   1:  PR[GP1:91,1] = PR[GP1:90,1] + -74.339;
   1:  PR[GP1:91,2] = PR[GP1:90,2] + 0.256;
   1:L PR[91] 10mm/sec CNT100;
   1:  PR[GP1:91,1] = PR[GP1:90,1] + -74.139;
   1:  PR[GP1:91,2] = PR[GP1:90,2] + -1.545;
   1:L PR[91] 10mm/sec CNT100;
   1:  PR[GP1:91,1] = PR[GP1:90,1] + -72.276;
   1:  PR[GP1:91,2] = PR[GP1:90,2] + -11.283;
   1:L PR[91] 10mm/sec CNT100;
   1:  PR[GP1:91,1] = PR[GP1:90,1] + -71.760;
   1:  PR[GP1:91,2] = PR[GP1:90,2] + -12.778;
   1:L PR[91] 10mm/sec CNT100;
   1:  PR[GP1:91,1] = PR[GP1:90,1] + -70.908;
   1:  PR[GP1:91,2] = PR[GP1:90,2] + -14.156;
   1:L PR[91] 10mm/sec CNT100;
   1:  PR[GP1:91,1] = PR[GP1:90,1] + -65.415;
   1:  PR[GP1:91,2] = PR[GP1:90,2] + -22.829;
   1:L PR[91] 10mm/sec CNT100;
   1:  PR[GP1:91,1] = PR[GP1:90,1] + -64.501;
   1:  PR[GP1:91,2] = PR[GP1:90,2] + -23.762;
   1:L PR[91] 10mm/sec CNT100;
   1:  PR[GP1:91,1] = PR[GP1:90,1] + -63.337;
   1:  PR[GP1:91,2] = PR[GP1:90,2] + -24.515;
   1:L PR[91] 10mm/sec CNT100;
   1:  PR[GP1:91,1] = PR[GP1:90,1] + -54.747;
   1:  PR[GP1:91,2] = PR[GP1:90,2] + -30.797;
   1:L PR[91] 10mm/sec CNT100;
   1:  PR[GP1:91,1] = PR[GP1:90,1] + -53.911;
   1:  PR[GP1:91,2] = PR[GP1:90,2] + -31.105;
   1:L PR[91] 10mm/sec CNT100;
   1:  PR[GP1:91,1] = PR[GP1:90,1] + -42.471;
   1:  PR[GP1:91,2] = PR[GP1:90,2] + -34.073;
   1:L PR[91] 10mm/sec CNT100;
   1:  PR[GP1:91,1] = PR[GP1:90,1] + -42.174;
   1:  PR[GP1:91,2] = PR[GP1:90,2] + -34.112;
   1:L PR[91] 10mm/sec CNT100;
   1:  PR[GP1:91,1] = PR[GP1:90,1] + -41.849;
   1:  PR[GP1:91,2] = PR[GP1:90,2] + -34.082;
   1:L PR[91] 10mm/sec CNT100;
   1:  PR[GP1:91,1] = PR[GP1:90,1] + -34.975;
   1:  PR[GP1:91,2] = PR[GP1:90,2] + -33.253;
   1:L PR[91] 10mm/sec CNT100;
   1:  PR[GP1:91,1] = PR[GP1:90,1] + -29.454;
   1:  PR[GP1:91,2] = PR[GP1:90,2] + -32.634;
   1:L PR[91] 10mm/sec CNT100;
   1:  PR[GP1:91,1] = PR[GP1:90,1] + -28.961;
   1:  PR[GP1:91,2] = PR[GP1:90,2] + -32.418;
   1:L PR[91] 10mm/sec CNT100;
   1:  PR[GP1:91,1] = PR[GP1:90,1] + -18.207;
   1:  PR[GP1:91,2] = PR[GP1:90,2] + -26.771;
   1:L PR[91] 10mm/sec CNT100;
   1:  PR[GP1:91,1] = PR[GP1:90,1] + -16.790;
   1:  PR[GP1:91,2] = PR[GP1:90,2] + -25.386;
   1:L PR[91] 10mm/sec CNT100;
   1:  PR[GP1:91,1] = PR[GP1:90,1] + -9.851;
   1:  PR[GP1:91,2] = PR[GP1:90,2] + -17.341;
   1:L PR[91] 10mm/sec CNT100;
   1:  PR[GP1:91,1] = PR[GP1:90,1] + -8.556;
   1:  PR[GP1:91,2] = PR[GP1:90,2] + -14.548;
   1:L PR[91] 10mm/sec CNT100;
   1:  PR[GP1:91,1] = PR[GP1:90,1] + -5.279;
   1:  PR[GP1:91,2] = PR[GP1:90,2] + -5.083;
   1:L PR[91] 10mm/sec CNT100;
   1:  PR[GP1:91,1] = PR[GP1:90,1] + 4.751;
   1:L PR[91] 10mm/sec CNT100;
   1:  PR[GP1:91,1] = PR[GP1:90,1] + 7.580;
   1:  PR[GP1:91,2] = PR[GP1:90,2] + -13.769;
   1:  PR[GP1:91,3] = PR[GP1:90,3] + 17.995;
   1:L PR[91] 10mm/sec CNT100;
   1:  PR[GP1:91,1] = PR[GP1:90,1] + 9.344;
   1:  PR[GP1:91,2] = PR[GP1:90,2] + -17.567;
   1:L PR[91] 10mm/sec CNT100;
   1:  PR[GP1:91,1] = PR[GP1:90,1] + 15.538;
   1:  PR[GP1:91,2] = PR[GP1:90,2] + -24.755;
   1:L PR[91] 10mm/sec CNT100;
   1:  PR[GP1:91,1] = PR[GP1:90,1] + 17.739;
   1:  PR[GP1:91,2] = PR[GP1:90,2] + -26.911;
   1:L PR[91] 10mm/sec CNT100;
   1:  PR[GP1:91,1] = PR[GP1:90,1] + 27.542;
   1:  PR[GP1:91,2] = PR[GP1:90,2] + -32.059;
   1:L PR[91] 10mm/sec CNT100;
   1:  PR[GP1:91,1] = PR[GP1:90,1] + 28.984;
   1:  PR[GP1:91,2] = PR[GP1:90,2] + -32.692;
   1:L PR[91] 10mm/sec CNT100;
   1:  PR[GP1:91,1] = PR[GP1:90,1] + 41.685;
   1:  PR[GP1:91,2] = PR[GP1:90,2] + -34.108;
   1:L PR[91] 10mm/sec CNT100;
   1:  PR[GP1:91,1] = PR[GP1:90,1] + 53.747;
   1:  PR[GP1:91,2] = PR[GP1:90,2] + -30.970;
   1:L PR[91] 10mm/sec CNT100;
   1:  PR[GP1:91,1] = PR[GP1:90,1] + 54.176;
   1:  PR[GP1:91,2] = PR[GP1:90,2] + -30.813;
   1:L PR[91] 10mm/sec CNT100;
   1:  PR[GP1:91,1] = PR[GP1:90,1] + 54.570;
   1:  PR[GP1:91,2] = PR[GP1:90,2] + -30.558;
   1:L PR[91] 10mm/sec CNT100;
   1:  PR[GP1:91,1] = PR[GP1:90,1] + 64.128;
   1:  PR[GP1:91,2] = PR[GP1:90,2] + -23.600;
   1:L PR[91] 10mm/sec CNT100;
   1:  PR[GP1:91,1] = PR[GP1:90,1] + 64.755;
   1:  PR[GP1:91,2] = PR[GP1:90,2] + -22.960;
   1:L PR[91] 10mm/sec CNT100;
   1:  PR[GP1:91,1] = PR[GP1:90,1] + 65.254;
   1:  PR[GP1:91,2] = PR[GP1:90,2] + -22.153;
   1:L PR[91] 10mm/sec CNT100;
   1:  PR[GP1:91,1] = PR[GP1:90,1] + 71.263;
   1:  PR[GP1:91,2] = PR[GP1:90,2] + -12.665;
   1:L PR[91] 10mm/sec CNT100;
   1:  PR[GP1:91,1] = PR[GP1:90,1] + 71.637;
   1:  PR[GP1:91,2] = PR[GP1:90,2] + -11.579;
   1:L PR[91] 10mm/sec CNT100;
   1:  PR[GP1:91,1] = PR[GP1:90,1] + 71.774;
   1:  PR[GP1:91,2] = PR[GP1:90,2] + -10.346;
   1:L PR[91] 10mm/sec CNT100;
   1:  PR[GP1:91,1] = PR[GP1:90,1] + 73.791;
   1:  PR[GP1:91,2] = PR[GP1:90,2] + 0.302;
   1:L PR[91] 10mm/sec CNT100;
   1:  PR[GP1:91,1] = PR[GP1:90,1] + 73.634;
   1:  PR[GP1:91,2] = PR[GP1:90,2] + 1.715;
   1:L PR[91] 10mm/sec CNT100;
   1:  PR[GP1:91,1] = PR[GP1:90,1] + 71.645;
   1:  PR[GP1:91,2] = PR[GP1:90,2] + 12.115;
   1:L PR[91] 10mm/sec CNT100;
   1:  PR[GP1:91,1] = PR[GP1:90,1] + 71.262;
   1:  PR[GP1:91,2] = PR[GP1:90,2] + 13.226;
   1:L PR[91] 10mm/sec CNT100;
   1:  PR[GP1:91,1] = PR[GP1:90,1] + 70.623;
   1:  PR[GP1:91,2] = PR[GP1:90,2] + 14.259;
   1:L PR[91] 10mm/sec CNT100;
   1:  PR[GP1:91,1] = PR[GP1:90,1] + 64.757;
   1:  PR[GP1:91,2] = PR[GP1:90,2] + 23.516;
   1:L PR[91] 10mm/sec CNT100;
   1:  PR[GP1:91,1] = PR[GP1:90,1] + 64.140;
   1:  PR[GP1:91,2] = PR[GP1:90,2] + 24.146;
   1:L PR[91] 10mm/sec CNT100;
   1:  PR[GP1:91,1] = PR[GP1:90,1] + 63.331;
   1:  PR[GP1:91,2] = PR[GP1:90,2] + 24.669;
   1:L PR[91] 10mm/sec CNT100;
   1:  PR[GP1:91,1] = PR[GP1:90,1] + 54.159;
   1:  PR[GP1:91,2] = PR[GP1:90,2] + 31.377;
   1:L PR[91] 10mm/sec CNT100;
   1:  PR[GP1:91,1] = PR[GP1:90,1] + 53.747;
   1:  PR[GP1:91,2] = PR[GP1:90,2] + 31.529;
   1:L PR[91] 10mm/sec CNT100;
   1:  PR[GP1:91,1] = PR[GP1:90,1] + 41.668;
   1:  PR[GP1:91,2] = PR[GP1:90,2] + 34.670;
   1:L PR[91] 10mm/sec CNT100;
   1:  PR[GP1:91,1] = PR[GP1:90,1] + 41.604;
   1:  PR[GP1:91,2] = PR[GP1:90,2] + 34.667;
   1:L PR[91] 10mm/sec CNT100;
   1:  PR[GP1:91,1] = PR[GP1:90,1] + 28.984;
   1:  PR[GP1:91,2] = PR[GP1:90,2] + 33.250;
   1:L PR[91] 10mm/sec CNT100;
   1:  PR[GP1:91,1] = PR[GP1:90,1] + 27.542;
   1:  PR[GP1:91,2] = PR[GP1:90,2] + 32.617;
   1:L PR[91] 10mm/sec CNT100;
   1:  PR[GP1:91,1] = PR[GP1:90,1] + 17.739;
   1:  PR[GP1:91,2] = PR[GP1:90,2] + 27.469;
   1:L PR[91] 10mm/sec CNT100;
   1:  PR[GP1:91,1] = PR[GP1:90,1] + 15.538;
   1:  PR[GP1:91,2] = PR[GP1:90,2] + 25.313;
   1:L PR[91] 10mm/sec CNT100;
   1:  PR[GP1:91,1] = PR[GP1:90,1] + 9.344;
   1:  PR[GP1:91,2] = PR[GP1:90,2] + 18.125;
   1:L PR[91] 10mm/sec CNT100;
   1:  PR[GP1:91,1] = PR[GP1:90,1] + 7.579;
   1:  PR[GP1:91,2] = PR[GP1:90,2] + 14.325;
   1:L PR[91] 10mm/sec CNT100;
   1:  PR[GP1:91,1] = PR[GP1:90,1] + 4.686;
   1:  PR[GP1:91,2] = PR[GP1:90,2] + 5.966;
   1:L PR[91] 10mm/sec CNT100;
   1:  PR[GP1:91,1] = PR[GP1:90,1] + -5.214;
   1:L PR[91] 10mm/sec CNT100;
   1:  PR[GP1:91,1] = PR[GP1:90,1] + -8.111;
   1:  PR[GP1:91,2] = PR[GP1:90,2] + 14.333;
   1:L PR[91] 10mm/sec CNT100;
   1:  PR[GP1:91,1] = PR[GP1:90,1] + -9.876;
   1:  PR[GP1:91,2] = PR[GP1:90,2] + 18.139;
   1:L PR[91] 10mm/sec CNT100;
   1:  PR[GP1:91,1] = PR[GP1:90,1] + -16.071;
   1:  PR[GP1:91,2] = PR[GP1:90,2] + 25.322;
   1:L PR[91] 10mm/sec CNT100;
   1:  PR[GP1:91,1] = PR[GP1:90,1] + -18.271;
   1:  PR[GP1:91,2] = PR[GP1:90,2] + 27.472;
   1:L PR[91] 10mm/sec CNT100;
   1:  PR[GP1:91,1] = PR[GP1:90,1] + -28.075;
   1:  PR[GP1:91,2] = PR[GP1:90,2] + 32.620;
   1:L PR[91] 10mm/sec CNT100;
   1:  PR[GP1:91,1] = PR[GP1:90,1] + -29.516;
   1:  PR[GP1:91,2] = PR[GP1:90,2] + 33.252;
   1:L PR[91] 10mm/sec CNT100;
   1:  PR[GP1:91,1] = PR[GP1:90,1] + -42.215;
   1:  PR[GP1:91,2] = PR[GP1:90,2] + 34.666;
   1:L PR[91] 10mm/sec CNT100;
   1:  PR[GP1:91,1] = PR[GP1:90,1] + -54.276;
   1:  PR[GP1:91,2] = PR[GP1:90,2] + 31.527;
   1:L PR[91] 10mm/sec CNT100;
   1:  PR[GP1:91,1] = PR[GP1:90,1] + -54.705;
   1:  PR[GP1:91,2] = PR[GP1:90,2] + 31.369;
   1:L PR[91] 10mm/sec CNT100;
   1:  PR[GP1:91,1] = PR[GP1:90,1] + -55.099;
   1:  PR[GP1:91,2] = PR[GP1:90,2] + 31.114;
   1:L PR[91] 10mm/sec CNT100;
   1:  PR[GP1:91,1] = PR[GP1:90,1] + -64.656;
   1:  PR[GP1:91,2] = PR[GP1:90,2] + 24.157;
   1:L PR[91] 10mm/sec CNT100;
   1:  PR[GP1:91,1] = PR[GP1:90,1] + -65.285;
   1:  PR[GP1:91,2] = PR[GP1:90,2] + 23.515;
   1:L PR[91] 10mm/sec CNT100;
   1:  PR[GP1:91,1] = PR[GP1:90,1] + -71.790;
   1:  PR[GP1:91,2] = PR[GP1:90,2] + 13.220;
   1:L PR[91] 10mm/sec CNT100;
   1:  PR[GP1:91,1] = PR[GP1:90,1] + -72.164;
   1:  PR[GP1:91,2] = PR[GP1:90,2] + 12.134;
   1:L PR[91] 10mm/sec CNT100;
   1:  PR[GP1:91,1] = PR[GP1:90,1] + -72.301;
   1:  PR[GP1:91,2] = PR[GP1:90,2] + 10.901;
   1:L PR[91] 10mm/sec CNT100;
   1:  PR[GP1:91,1] = PR[GP1:90,1] + -74.318;
   1:  PR[GP1:91,2] = PR[GP1:90,2] + 0.256;
   1:L PR[91] 10mm/sec CNT100;
   1:  PR[GP1:91,1] = PR[GP1:90,1] + -74.160;
   1:  PR[GP1:91,2] = PR[GP1:90,2] + -1.157;
   1:L PR[91] 10mm/sec CNT100;
   1:  PR[GP1:91,1] = PR[GP1:90,1] + -72.172;
   1:  PR[GP1:91,2] = PR[GP1:90,2] + -11.554;
   1:L PR[91] 10mm/sec CNT100;
   1:  PR[GP1:91,1] = PR[GP1:90,1] + -71.789;
   1:  PR[GP1:91,2] = PR[GP1:90,2] + -12.665;
   1:L PR[91] 10mm/sec CNT100;
   1:  PR[GP1:91,1] = PR[GP1:90,1] + -71.150;
   1:  PR[GP1:91,2] = PR[GP1:90,2] + -13.698;
   1:L PR[91] 10mm/sec CNT100;
   1:  PR[GP1:91,1] = PR[GP1:90,1] + -65.285;
   1:  PR[GP1:91,2] = PR[GP1:90,2] + -22.957;
   1:L PR[91] 10mm/sec CNT100;
   1:  PR[GP1:91,1] = PR[GP1:90,1] + -64.667;
   1:  PR[GP1:91,2] = PR[GP1:90,2] + -23.587;
   1:L PR[91] 10mm/sec CNT100;
   1:  PR[GP1:91,1] = PR[GP1:90,1] + -63.859;
   1:  PR[GP1:91,2] = PR[GP1:90,2] + -24.110;
   1:L PR[91] 10mm/sec CNT100;
   1:  PR[GP1:91,1] = PR[GP1:90,1] + -54.688;
   1:  PR[GP1:91,2] = PR[GP1:90,2] + -30.818;
   1:L PR[91] 10mm/sec CNT100;
   1:  PR[GP1:91,1] = PR[GP1:90,1] + -54.276;
   1:  PR[GP1:91,2] = PR[GP1:90,2] + -30.969;
   1:L PR[91] 10mm/sec CNT100;
   1:  PR[GP1:91,1] = PR[GP1:90,1] + -42.215;
   1:  PR[GP1:91,2] = PR[GP1:90,2] + -34.107;
   1:L PR[91] 10mm/sec CNT100;
   1:  PR[GP1:91,1] = PR[GP1:90,1] + -29.516;
   1:  PR[GP1:91,2] = PR[GP1:90,2] + -32.694;
   1:L PR[91] 10mm/sec CNT100;
   1:  PR[GP1:91,1] = PR[GP1:90,1] + -28.075;
   1:  PR[GP1:91,2] = PR[GP1:90,2] + -32.062;
   1:L PR[91] 10mm/sec CNT100;
   1:  PR[GP1:91,1] = PR[GP1:90,1] + -18.271;
   1:  PR[GP1:91,2] = PR[GP1:90,2] + -26.914;
   1:L PR[91] 10mm/sec CNT100;
   1:  PR[GP1:91,1] = PR[GP1:90,1] + -16.071;
   1:  PR[GP1:91,2] = PR[GP1:90,2] + -24.763;
   1:L PR[91] 10mm/sec CNT100;
   1:  PR[GP1:91,1] = PR[GP1:90,1] + -9.876;
   1:  PR[GP1:91,2] = PR[GP1:90,2] + -17.581;
   1:L PR[91] 10mm/sec CNT100;
   1:  PR[GP1:91,1] = PR[GP1:90,1] + -8.110;
   1:  PR[GP1:91,2] = PR[GP1:90,2] + -13.773;
   1:L PR[91] 10mm/sec CNT100;
   1:  PR[GP1:91,1] = PR[GP1:90,1] + -5.214;
   1:  PR[GP1:91,2] = PR[GP1:90,2] + -5.408;
   1:L PR[91] 10mm/sec CNT100;
   1:  PR[GP1:91,1] = PR[GP1:90,1] + 4.686;
   1:L PR[91] 10mm/sec CNT100;
   1:  PR[GP1:91,1] = PR[GP1:90,1] + 7.134;
   1:  PR[GP1:91,2] = PR[GP1:90,2] + -12.995;
   1:  PR[GP1:91,3] = PR[GP1:90,3] + 18.605;
   1:L PR[91] 10mm/sec CNT100;
   1:  PR[GP1:91,1] = PR[GP1:90,1] + 9.368;
   1:  PR[GP1:91,2] = PR[GP1:90,2] + -17.806;
   1:L PR[91] 10mm/sec CNT100;
   1:  PR[GP1:91,1] = PR[GP1:90,1] + 14.818;
   1:  PR[GP1:91,2] = PR[GP1:90,2] + -24.130;
   1:L PR[91] 10mm/sec CNT100;
   1:  PR[GP1:91,1] = PR[GP1:90,1] + 17.802;
   1:  PR[GP1:91,2] = PR[GP1:90,2] + -27.054;
   1:L PR[91] 10mm/sec CNT100;
   1:  PR[GP1:91,1] = PR[GP1:90,1] + 26.655;
   1:  PR[GP1:91,2] = PR[GP1:90,2] + -31.703;
   1:L PR[91] 10mm/sec CNT100;
   1:  PR[GP1:91,1] = PR[GP1:90,1] + 29.045;
   1:  PR[GP1:91,2] = PR[GP1:90,2] + -32.752;
   1:L PR[91] 10mm/sec CNT100;
   1:  PR[GP1:91,1] = PR[GP1:90,1] + 40.686;
   1:  PR[GP1:91,2] = PR[GP1:90,2] + -34.059;
   1:L PR[91] 10mm/sec CNT100;
   1:  PR[GP1:91,1] = PR[GP1:90,1] + 41.701;
   1:  PR[GP1:91,2] = PR[GP1:90,2] + -34.116;
   1:L PR[91] 10mm/sec CNT100;
   1:  PR[GP1:91,1] = PR[GP1:90,1] + 54.124;
   1:  PR[GP1:91,2] = PR[GP1:90,2] + -30.822;
   1:L PR[91] 10mm/sec CNT100;
   1:  PR[GP1:91,1] = PR[GP1:90,1] + 64.295;
   1:  PR[GP1:91,2] = PR[GP1:90,2] + -23.426;
   1:L PR[91] 10mm/sec CNT100;
   1:  PR[GP1:91,1] = PR[GP1:90,1] + 64.627;
   1:  PR[GP1:91,2] = PR[GP1:90,2] + -23.086;
   1:L PR[91] 10mm/sec CNT100;
   1:  PR[GP1:91,1] = PR[GP1:90,1] + 71.291;
   1:  PR[GP1:91,2] = PR[GP1:90,2] + -12.552;
   1:L PR[91] 10mm/sec CNT100;
   1:  PR[GP1:91,1] = PR[GP1:90,1] + 71.533;
   1:  PR[GP1:91,2] = PR[GP1:90,2] + -11.850;
   1:L PR[91] 10mm/sec CNT100;
   1:  PR[GP1:91,1] = PR[GP1:90,1] + 71.625;
   1:  PR[GP1:91,2] = PR[GP1:90,2] + -11.021;
   1:L PR[91] 10mm/sec CNT100;
   1:  PR[GP1:91,1] = PR[GP1:90,1] + 73.770;
   1:  PR[GP1:91,2] = PR[GP1:90,2] + 0.302;
   1:L PR[91] 10mm/sec CNT100;
   1:  PR[GP1:91,1] = PR[GP1:90,1] + 73.656;
   1:  PR[GP1:91,2] = PR[GP1:90,2] + 1.327;
   1:L PR[91] 10mm/sec CNT100;
   1:  PR[GP1:91,1] = PR[GP1:90,1] + 71.541;
   1:  PR[GP1:91,2] = PR[GP1:90,2] + 12.386;
   1:L PR[91] 10mm/sec CNT100;
   1:  PR[GP1:91,1] = PR[GP1:90,1] + 71.291;
   1:  PR[GP1:91,2] = PR[GP1:90,2] + 13.110;
   1:L PR[91] 10mm/sec CNT100;
   1:  PR[GP1:91,1] = PR[GP1:90,1] + 64.627;
   1:  PR[GP1:91,2] = PR[GP1:90,2] + 23.644;
   1:L PR[91] 10mm/sec CNT100;
   1:  PR[GP1:91,1] = PR[GP1:90,1] + 64.306;
   1:  PR[GP1:91,2] = PR[GP1:90,2] + 23.972;
   1:L PR[91] 10mm/sec CNT100;
   1:  PR[GP1:91,1] = PR[GP1:90,1] + 63.853;
   1:  PR[GP1:91,2] = PR[GP1:90,2] + 24.265;
   1:L PR[91] 10mm/sec CNT100;
   1:  PR[GP1:91,1] = PR[GP1:90,1] + 54.123;
   1:  PR[GP1:91,2] = PR[GP1:90,2] + 31.380;
   1:L PR[91] 10mm/sec CNT100;
   1:  PR[GP1:91,1] = PR[GP1:90,1] + 41.701;
   1:  PR[GP1:91,2] = PR[GP1:90,2] + 34.674;
   1:L PR[91] 10mm/sec CNT100;
   1:  PR[GP1:91,1] = PR[GP1:90,1] + 40.686;
   1:  PR[GP1:91,2] = PR[GP1:90,2] + 34.617;
   1:L PR[91] 10mm/sec CNT100;
   1:  PR[GP1:91,1] = PR[GP1:90,1] + 29.045;
   1:  PR[GP1:91,2] = PR[GP1:90,2] + 33.310;
   1:L PR[91] 10mm/sec CNT100;
   1:  PR[GP1:91,1] = PR[GP1:90,1] + 26.655;
   1:  PR[GP1:91,2] = PR[GP1:90,2] + 32.261;
   1:L PR[91] 10mm/sec CNT100;
   1:  PR[GP1:91,1] = PR[GP1:90,1] + 17.802;
   1:  PR[GP1:91,2] = PR[GP1:90,2] + 27.612;
   1:L PR[91] 10mm/sec CNT100;
   1:  PR[GP1:91,1] = PR[GP1:90,1] + 14.818;
   1:  PR[GP1:91,2] = PR[GP1:90,2] + 24.688;
   1:L PR[91] 10mm/sec CNT100;
   1:  PR[GP1:91,1] = PR[GP1:90,1] + 9.368;
   1:  PR[GP1:91,2] = PR[GP1:90,2] + 18.364;
   1:L PR[91] 10mm/sec CNT100;
   1:  PR[GP1:91,1] = PR[GP1:90,1] + 7.133;
   1:  PR[GP1:91,2] = PR[GP1:90,2] + 13.550;
   1:L PR[91] 10mm/sec CNT100;
   1:  PR[GP1:91,1] = PR[GP1:90,1] + 4.620;
   1:  PR[GP1:91,2] = PR[GP1:90,2] + 6.291;
   1:L PR[91] 10mm/sec CNT100;
   1:  PR[GP1:91,1] = PR[GP1:90,1] + -5.149;
   1:L PR[91] 10mm/sec CNT100;
   1:  PR[GP1:91,1] = PR[GP1:90,1] + -7.665;
   1:  PR[GP1:91,2] = PR[GP1:90,2] + 13.559;
   1:L PR[91] 10mm/sec CNT100;
   1:  PR[GP1:91,1] = PR[GP1:90,1] + -9.901;
   1:  PR[GP1:91,2] = PR[GP1:90,2] + 18.379;
   1:L PR[91] 10mm/sec CNT100;
   1:  PR[GP1:91,1] = PR[GP1:90,1] + -15.352;
   1:  PR[GP1:91,2] = PR[GP1:90,2] + 24.699;
   1:L PR[91] 10mm/sec CNT100;
   1:  PR[GP1:91,1] = PR[GP1:90,1] + -18.335;
   1:  PR[GP1:91,2] = PR[GP1:90,2] + 27.615;
   1:L PR[91] 10mm/sec CNT100;
   1:  PR[GP1:91,1] = PR[GP1:90,1] + -27.189;
   1:  PR[GP1:91,2] = PR[GP1:90,2] + 32.264;
   1:L PR[91] 10mm/sec CNT100;
   1:  PR[GP1:91,1] = PR[GP1:90,1] + -29.577;
   1:  PR[GP1:91,2] = PR[GP1:90,2] + 33.313;
   1:L PR[91] 10mm/sec CNT100;
   1:  PR[GP1:91,1] = PR[GP1:90,1] + -41.217;
   1:  PR[GP1:91,2] = PR[GP1:90,2] + 34.617;
   1:L PR[91] 10mm/sec CNT100;
   1:  PR[GP1:91,1] = PR[GP1:90,1] + -42.231;
   1:  PR[GP1:91,2] = PR[GP1:90,2] + 34.673;
   1:L PR[91] 10mm/sec CNT100;
   1:  PR[GP1:91,1] = PR[GP1:90,1] + -54.653;
   1:  PR[GP1:91,2] = PR[GP1:90,2] + 31.379;
   1:L PR[91] 10mm/sec CNT100;
   1:  PR[GP1:91,1] = PR[GP1:90,1] + -64.822;
   1:  PR[GP1:91,2] = PR[GP1:90,2] + 23.983;
   1:L PR[91] 10mm/sec CNT100;
   1:  PR[GP1:91,1] = PR[GP1:90,1] + -65.155;
   1:  PR[GP1:91,2] = PR[GP1:90,2] + 23.643;
   1:L PR[91] 10mm/sec CNT100;
   1:  PR[GP1:91,1] = PR[GP1:90,1] + -71.818;
   1:  PR[GP1:91,2] = PR[GP1:90,2] + 13.107;
   1:L PR[91] 10mm/sec CNT100;
   1:  PR[GP1:91,1] = PR[GP1:90,1] + -72.060;
   1:  PR[GP1:91,2] = PR[GP1:90,2] + 12.405;
   1:L PR[91] 10mm/sec CNT100;
   1:  PR[GP1:91,1] = PR[GP1:90,1] + -72.152;
   1:  PR[GP1:91,2] = PR[GP1:90,2] + 11.575;
   1:L PR[91] 10mm/sec CNT100;
   1:  PR[GP1:91,1] = PR[GP1:90,1] + -74.296;
   1:  PR[GP1:91,2] = PR[GP1:90,2] + 0.256;
   1:L PR[91] 10mm/sec CNT100;
   1:  PR[GP1:91,1] = PR[GP1:90,1] + -74.182;
   1:  PR[GP1:91,2] = PR[GP1:90,2] + -0.769;
   1:L PR[91] 10mm/sec CNT100;
   1:  PR[GP1:91,1] = PR[GP1:90,1] + -72.067;
   1:  PR[GP1:91,2] = PR[GP1:90,2] + -11.825;
   1:L PR[91] 10mm/sec CNT100;
   1:  PR[GP1:91,1] = PR[GP1:90,1] + -71.817;
   1:  PR[GP1:91,2] = PR[GP1:90,2] + -12.551;
   1:L PR[91] 10mm/sec CNT100;
   1:  PR[GP1:91,1] = PR[GP1:90,1] + -71.392;
   1:  PR[GP1:91,2] = PR[GP1:90,2] + -13.239;
   1:L PR[91] 10mm/sec CNT100;
   1:  PR[GP1:91,1] = PR[GP1:90,1] + -65.155;
   1:  PR[GP1:91,2] = PR[GP1:90,2] + -23.085;
   1:L PR[91] 10mm/sec CNT100;
   1:  PR[GP1:91,1] = PR[GP1:90,1] + -64.834;
   1:  PR[GP1:91,2] = PR[GP1:90,2] + -23.413;
   1:L PR[91] 10mm/sec CNT100;
   1:  PR[GP1:91,1] = PR[GP1:90,1] + -64.381;
   1:  PR[GP1:91,2] = PR[GP1:90,2] + -23.706;
   1:L PR[91] 10mm/sec CNT100;
   1:  PR[GP1:91,1] = PR[GP1:90,1] + -54.632;
   1:  PR[GP1:91,2] = PR[GP1:90,2] + -30.836;
   1:L PR[91] 10mm/sec CNT100;
   1:  PR[GP1:91,1] = PR[GP1:90,1] + -42.232;
   1:  PR[GP1:91,2] = PR[GP1:90,2] + -34.115;
   1:L PR[91] 10mm/sec CNT100;
   1:  PR[GP1:91,1] = PR[GP1:90,1] + -41.217;
   1:  PR[GP1:91,2] = PR[GP1:90,2] + -34.059;
   1:L PR[91] 10mm/sec CNT100;
   1:  PR[GP1:91,1] = PR[GP1:90,1] + -29.577;
   1:  PR[GP1:91,2] = PR[GP1:90,2] + -32.755;
   1:L PR[91] 10mm/sec CNT100;
   1:  PR[GP1:91,1] = PR[GP1:90,1] + -27.189;
   1:  PR[GP1:91,2] = PR[GP1:90,2] + -31.706;
   1:L PR[91] 10mm/sec CNT100;
   1:  PR[GP1:91,1] = PR[GP1:90,1] + -18.335;
   1:  PR[GP1:91,2] = PR[GP1:90,2] + -27.057;
   1:L PR[91] 10mm/sec CNT100;
   1:  PR[GP1:91,1] = PR[GP1:90,1] + -15.351;
   1:  PR[GP1:91,2] = PR[GP1:90,2] + -24.141;
   1:L PR[91] 10mm/sec CNT100;
   1:  PR[GP1:91,1] = PR[GP1:90,1] + -9.901;
   1:  PR[GP1:91,2] = PR[GP1:90,2] + -17.821;
   1:L PR[91] 10mm/sec CNT100;
   1:  PR[GP1:91,1] = PR[GP1:90,1] + -7.664;
   1:  PR[GP1:91,2] = PR[GP1:90,2] + -12.997;
   1:L PR[91] 10mm/sec CNT100;
   1:  PR[GP1:91,1] = PR[GP1:90,1] + -5.149;
   1:  PR[GP1:91,2] = PR[GP1:90,2] + -5.733;
   1:L PR[91] 10mm/sec CNT100;
   1:  PR[GP1:91,1] = PR[GP1:90,1] + 4.620;
   1:L PR[91] 10mm/sec CNT100;
   1:  PR[GP1:91,1] = PR[GP1:90,1] + 6.689;
   1:  PR[GP1:91,2] = PR[GP1:90,2] + -12.221;
   1:  PR[GP1:91,3] = PR[GP1:90,3] + 19.215;
   1:L PR[91] 10mm/sec CNT100;
   1:  PR[GP1:91,1] = PR[GP1:90,1] + 9.392;
   1:  PR[GP1:91,2] = PR[GP1:90,2] + -18.045;
   1:L PR[91] 10mm/sec CNT100;
   1:  PR[GP1:91,1] = PR[GP1:90,1] + 14.098;
   1:  PR[GP1:91,2] = PR[GP1:90,2] + -23.505;
   1:L PR[91] 10mm/sec CNT100;
   1:  PR[GP1:91,1] = PR[GP1:90,1] + 17.865;
   1:  PR[GP1:91,2] = PR[GP1:90,2] + -27.197;
   1:L PR[91] 10mm/sec CNT100;
   1:  PR[GP1:91,1] = PR[GP1:90,1] + 25.768;
   1:  PR[GP1:91,2] = PR[GP1:90,2] + -31.346;
   1:L PR[91] 10mm/sec CNT100;
   1:  PR[GP1:91,1] = PR[GP1:90,1] + 29.106;
   1:  PR[GP1:91,2] = PR[GP1:90,2] + -32.812;
   1:L PR[91] 10mm/sec CNT100;
   1:  PR[GP1:91,1] = PR[GP1:90,1] + 39.767;
   1:  PR[GP1:91,2] = PR[GP1:90,2] + -34.009;
   1:L PR[91] 10mm/sec CNT100;
   1:  PR[GP1:91,1] = PR[GP1:90,1] + 41.734;
   1:  PR[GP1:91,2] = PR[GP1:90,2] + -34.119;
   1:L PR[91] 10mm/sec CNT100;
   1:  PR[GP1:91,1] = PR[GP1:90,1] + 53.561;
   1:  PR[GP1:91,2] = PR[GP1:90,2] + -30.982;
   1:L PR[91] 10mm/sec CNT100;
   1:  PR[GP1:91,1] = PR[GP1:90,1] + 54.098;
   1:  PR[GP1:91,2] = PR[GP1:90,2] + -30.815;
   1:L PR[91] 10mm/sec CNT100;
   1:  PR[GP1:91,1] = PR[GP1:90,1] + 64.461;
   1:  PR[GP1:91,2] = PR[GP1:90,2] + -23.252;
   1:L PR[91] 10mm/sec CNT100;
   1:  PR[GP1:91,1] = PR[GP1:90,1] + 64.498;
   1:  PR[GP1:91,2] = PR[GP1:90,2] + -23.214;
   1:L PR[91] 10mm/sec CNT100;
   1:  PR[GP1:91,1] = PR[GP1:90,1] + 71.319;
   1:  PR[GP1:91,2] = PR[GP1:90,2] + -12.439;
   1:L PR[91] 10mm/sec CNT100;
   1:  PR[GP1:91,1] = PR[GP1:90,1] + 71.429;
   1:  PR[GP1:91,2] = PR[GP1:90,2] + -12.121;
   1:L PR[91] 10mm/sec CNT100;
   1:  PR[GP1:91,1] = PR[GP1:90,1] + 71.476;
   1:  PR[GP1:91,2] = PR[GP1:90,2] + -11.695;
   1:L PR[91] 10mm/sec CNT100;
   1:  PR[GP1:91,1] = PR[GP1:90,1] + 73.748;
   1:  PR[GP1:91,2] = PR[GP1:90,2] + 0.302;
   1:L PR[91] 10mm/sec CNT100;
   1:  PR[GP1:91,1] = PR[GP1:90,1] + 73.678;
   1:  PR[GP1:91,2] = PR[GP1:90,2] + 0.939;
   1:L PR[91] 10mm/sec CNT100;
   1:  PR[GP1:91,1] = PR[GP1:90,1] + 71.437;
   1:  PR[GP1:91,2] = PR[GP1:90,2] + 12.657;
   1:L PR[91] 10mm/sec CNT100;
   1:  PR[GP1:91,1] = PR[GP1:90,1] + 71.318;
   1:  PR[GP1:91,2] = PR[GP1:90,2] + 13.000;
   1:L PR[91] 10mm/sec CNT100;
   1:  PR[GP1:91,1] = PR[GP1:90,1] + 71.107;
   1:  PR[GP1:91,2] = PR[GP1:90,2] + 13.342;
   1:L PR[91] 10mm/sec CNT100;
   1:  PR[GP1:91,1] = PR[GP1:90,1] + 64.498;
   1:  PR[GP1:91,2] = PR[GP1:90,2] + 23.772;
   1:L PR[91] 10mm/sec CNT100;
   1:  PR[GP1:91,1] = PR[GP1:90,1] + 64.461;
   1:  PR[GP1:91,2] = PR[GP1:90,2] + 23.810;
   1:L PR[91] 10mm/sec CNT100;
   1:  PR[GP1:91,1] = PR[GP1:90,1] + 54.098;
   1:  PR[GP1:91,2] = PR[GP1:90,2] + 31.373;
   1:L PR[91] 10mm/sec CNT100;
   1:  PR[GP1:91,1] = PR[GP1:90,1] + 53.561;
   1:  PR[GP1:91,2] = PR[GP1:90,2] + 31.540;
   1:L PR[91] 10mm/sec CNT100;
   1:  PR[GP1:91,1] = PR[GP1:90,1] + 41.734;
   1:  PR[GP1:91,2] = PR[GP1:90,2] + 34.677;
   1:L PR[91] 10mm/sec CNT100;
   1:  PR[GP1:91,1] = PR[GP1:90,1] + 39.767;
   1:  PR[GP1:91,2] = PR[GP1:90,2] + 34.567;
   1:L PR[91] 10mm/sec CNT100;
   1:  PR[GP1:91,1] = PR[GP1:90,1] + 29.106;
   1:  PR[GP1:91,2] = PR[GP1:90,2] + 33.370;
   1:L PR[91] 10mm/sec CNT100;
   1:  PR[GP1:91,1] = PR[GP1:90,1] + 25.768;
   1:  PR[GP1:91,2] = PR[GP1:90,2] + 31.904;
   1:L PR[91] 10mm/sec CNT100;
   1:  PR[GP1:91,1] = PR[GP1:90,1] + 17.865;
   1:  PR[GP1:91,2] = PR[GP1:90,2] + 27.755;
   1:L PR[91] 10mm/sec CNT100;
   1:  PR[GP1:91,1] = PR[GP1:90,1] + 14.098;
   1:  PR[GP1:91,2] = PR[GP1:90,2] + 24.063;
   1:L PR[91] 10mm/sec CNT100;
   1:  PR[GP1:91,1] = PR[GP1:90,1] + 9.392;
   1:  PR[GP1:91,2] = PR[GP1:90,2] + 18.603;
   1:L PR[91] 10mm/sec CNT100;
   1:  PR[GP1:91,1] = PR[GP1:90,1] + 6.687;
   1:  PR[GP1:91,2] = PR[GP1:90,2] + 12.775;
   1:L PR[91] 10mm/sec CNT100;
   1:  PR[GP1:91,1] = PR[GP1:90,1] + 4.555;
   1:  PR[GP1:91,2] = PR[GP1:90,2] + 6.616;
   1:L PR[91] 10mm/sec CNT100;
   1:  PR[GP1:91,1] = PR[GP1:90,1] + -5.084;
   1:L PR[91] 10mm/sec CNT100;
   1:  PR[GP1:91,1] = PR[GP1:90,1] + -7.219;
   1:  PR[GP1:91,2] = PR[GP1:90,2] + 12.784;
   1:L PR[91] 10mm/sec CNT100;
   1:  PR[GP1:91,1] = PR[GP1:90,1] + -9.925;
   1:  PR[GP1:91,2] = PR[GP1:90,2] + 18.619;
   1:L PR[91] 10mm/sec CNT100;
   1:  PR[GP1:91,1] = PR[GP1:90,1] + -14.632;
   1:  PR[GP1:91,2] = PR[GP1:90,2] + 24.076;
   1:L PR[91] 10mm/sec CNT100;
   1:  PR[GP1:91,1] = PR[GP1:90,1] + -18.399;
   1:  PR[GP1:91,2] = PR[GP1:90,2] + 27.758;
   1:L PR[91] 10mm/sec CNT100;
   1:  PR[GP1:91,1] = PR[GP1:90,1] + -26.303;
   1:  PR[GP1:91,2] = PR[GP1:90,2] + 31.908;
   1:L PR[91] 10mm/sec CNT100;
   1:  PR[GP1:91,1] = PR[GP1:90,1] + -29.639;
   1:  PR[GP1:91,2] = PR[GP1:90,2] + 33.373;
   1:L PR[91] 10mm/sec CNT100;
   1:  PR[GP1:91,1] = PR[GP1:90,1] + -40.299;
   1:  PR[GP1:91,2] = PR[GP1:90,2] + 34.567;
   1:L PR[91] 10mm/sec CNT100;
   1:  PR[GP1:91,1] = PR[GP1:90,1] + -42.266;
   1:  PR[GP1:91,2] = PR[GP1:90,2] + 34.677;
   1:L PR[91] 10mm/sec CNT100;
   1:  PR[GP1:91,1] = PR[GP1:90,1] + -54.091;
   1:  PR[GP1:91,2] = PR[GP1:90,2] + 31.539;
   1:L PR[91] 10mm/sec CNT100;
   1:  PR[GP1:91,1] = PR[GP1:90,1] + -54.627;
   1:  PR[GP1:91,2] = PR[GP1:90,2] + 31.372;
   1:L PR[91] 10mm/sec CNT100;
   1:  PR[GP1:91,1] = PR[GP1:90,1] + -64.988;
   1:  PR[GP1:91,2] = PR[GP1:90,2] + 23.809;
   1:L PR[91] 10mm/sec CNT100;
   1:  PR[GP1:91,1] = PR[GP1:90,1] + -65.025;
   1:  PR[GP1:91,2] = PR[GP1:90,2] + 23.771;
   1:L PR[91] 10mm/sec CNT100;
   1:  PR[GP1:91,1] = PR[GP1:90,1] + -71.846;
   1:  PR[GP1:91,2] = PR[GP1:90,2] + 12.993;
   1:L PR[91] 10mm/sec CNT100;
   1:  PR[GP1:91,1] = PR[GP1:90,1] + -71.956;
   1:  PR[GP1:91,2] = PR[GP1:90,2] + 12.676;
   1:L PR[91] 10mm/sec CNT100;
   1:  PR[GP1:91,1] = PR[GP1:90,1] + -72.003;
   1:  PR[GP1:91,2] = PR[GP1:90,2] + 12.250;
   1:L PR[91] 10mm/sec CNT100;
   1:  PR[GP1:91,1] = PR[GP1:90,1] + -74.275;
   1:  PR[GP1:91,2] = PR[GP1:90,2] + 0.256;
   1:L PR[91] 10mm/sec CNT100;
   1:  PR[GP1:91,1] = PR[GP1:90,1] + -74.204;
   1:  PR[GP1:91,2] = PR[GP1:90,2] + -0.381;
   1:L PR[91] 10mm/sec CNT100;
   1:  PR[GP1:91,1] = PR[GP1:90,1] + -71.963;
   1:  PR[GP1:91,2] = PR[GP1:90,2] + -12.095;
   1:L PR[91] 10mm/sec CNT100;
   1:  PR[GP1:91,1] = PR[GP1:90,1] + -71.845;
   1:  PR[GP1:91,2] = PR[GP1:90,2] + -12.438;
   1:L PR[91] 10mm/sec CNT100;
   1:  PR[GP1:91,1] = PR[GP1:90,1] + -71.633;
   1:  PR[GP1:91,2] = PR[GP1:90,2] + -12.781;
   1:L PR[91] 10mm/sec CNT100;
   1:  PR[GP1:91,1] = PR[GP1:90,1] + -65.025;
   1:  PR[GP1:91,2] = PR[GP1:90,2] + -23.213;
   1:L PR[91] 10mm/sec CNT100;
   1:  PR[GP1:91,1] = PR[GP1:90,1] + -64.988;
   1:  PR[GP1:91,2] = PR[GP1:90,2] + -23.251;
   1:L PR[91] 10mm/sec CNT100;
   1:  PR[GP1:91,1] = PR[GP1:90,1] + -54.627;
   1:  PR[GP1:91,2] = PR[GP1:90,2] + -30.814;
   1:L PR[91] 10mm/sec CNT100;
   1:  PR[GP1:91,1] = PR[GP1:90,1] + -54.091;
   1:  PR[GP1:91,2] = PR[GP1:90,2] + -30.981;
   1:L PR[91] 10mm/sec CNT100;
   1:  PR[GP1:91,1] = PR[GP1:90,1] + -42.266;
   1:  PR[GP1:91,2] = PR[GP1:90,2] + -34.119;
   1:L PR[91] 10mm/sec CNT100;
   1:  PR[GP1:91,1] = PR[GP1:90,1] + -40.299;
   1:  PR[GP1:91,2] = PR[GP1:90,2] + -34.009;
   1:L PR[91] 10mm/sec CNT100;
   1:  PR[GP1:91,1] = PR[GP1:90,1] + -29.639;
   1:  PR[GP1:91,2] = PR[GP1:90,2] + -32.815;
   1:L PR[91] 10mm/sec CNT100;
   1:  PR[GP1:91,1] = PR[GP1:90,1] + -26.303;
   1:  PR[GP1:91,2] = PR[GP1:90,2] + -31.350;
   1:L PR[91] 10mm/sec CNT100;
   1:  PR[GP1:91,1] = PR[GP1:90,1] + -18.399;
   1:  PR[GP1:91,2] = PR[GP1:90,2] + -27.200;
   1:L PR[91] 10mm/sec CNT100;
   1:  PR[GP1:91,1] = PR[GP1:90,1] + -14.632;
   1:  PR[GP1:91,2] = PR[GP1:90,2] + -23.518;
   1:L PR[91] 10mm/sec CNT100;
   1:  PR[GP1:91,1] = PR[GP1:90,1] + -9.925;
   1:  PR[GP1:91,2] = PR[GP1:90,2] + -18.061;
   1:L PR[91] 10mm/sec CNT100;
   1:  PR[GP1:91,1] = PR[GP1:90,1] + -7.218;
   1:  PR[GP1:91,2] = PR[GP1:90,2] + -12.222;
   1:L PR[91] 10mm/sec CNT100;
   1:  PR[GP1:91,1] = PR[GP1:90,1] + -5.084;
   1:  PR[GP1:91,2] = PR[GP1:90,2] + -6.058;
   1:L PR[91] 10mm/sec CNT100;
   1:  PR[GP1:91,1] = PR[GP1:90,1] + 4.555;
   1:L PR[91] 10mm/sec CNT100;
   1:  PR[GP1:91,1] = PR[GP1:90,1] + 6.243;
   1:  PR[GP1:91,2] = PR[GP1:90,2] + -11.447;
   1:  PR[GP1:91,3] = PR[GP1:90,3] + 19.825;
   1:L PR[91] 10mm/sec CNT100;
   1:  PR[GP1:91,1] = PR[GP1:90,1] + 9.417;
   1:  PR[GP1:91,2] = PR[GP1:90,2] + -18.283;
   1:L PR[91] 10mm/sec CNT100;
   1:  PR[GP1:91,1] = PR[GP1:90,1] + 13.378;
   1:  PR[GP1:91,2] = PR[GP1:90,2] + -22.880;
   1:L PR[91] 10mm/sec CNT100;
   1:  PR[GP1:91,1] = PR[GP1:90,1] + 17.929;
   1:  PR[GP1:91,2] = PR[GP1:90,2] + -27.339;
   1:L PR[91] 10mm/sec CNT100;
   1:  PR[GP1:91,1] = PR[GP1:90,1] + 24.881;
   1:  PR[GP1:91,2] = PR[GP1:90,2] + -30.990;
   1:L PR[91] 10mm/sec CNT100;
   1:  PR[GP1:91,1] = PR[GP1:90,1] + 29.167;
   1:  PR[GP1:91,2] = PR[GP1:90,2] + -32.872;
   1:L PR[91] 10mm/sec CNT100;
   1:  PR[GP1:91,1] = PR[GP1:90,1] + 38.848;
   1:  PR[GP1:91,2] = PR[GP1:90,2] + -33.959;
   1:L PR[91] 10mm/sec CNT100;
   1:  PR[GP1:91,1] = PR[GP1:90,1] + 41.768;
   1:  PR[GP1:91,2] = PR[GP1:90,2] + -34.123;
   1:L PR[91] 10mm/sec CNT100;
   1:  PR[GP1:91,1] = PR[GP1:90,1] + 52.731;
   1:  PR[GP1:91,2] = PR[GP1:90,2] + -31.215;
   1:L PR[91] 10mm/sec CNT100;
   1:  PR[GP1:91,1] = PR[GP1:90,1] + 54.096;
   1:  PR[GP1:91,2] = PR[GP1:90,2] + -30.790;
   1:L PR[91] 10mm/sec CNT100;
   1:  PR[GP1:91,1] = PR[GP1:90,1] + 64.159;
   1:  PR[GP1:91,2] = PR[GP1:90,2] + -23.435;
   1:L PR[91] 10mm/sec CNT100;
   1:  PR[GP1:91,1] = PR[GP1:90,1] + 64.447;
   1:  PR[GP1:91,2] = PR[GP1:90,2] + -23.211;
   1:L PR[91] 10mm/sec CNT100;
   1:  PR[GP1:91,1] = PR[GP1:90,1] + 71.324;
   1:  PR[GP1:91,2] = PR[GP1:90,2] + -12.363;
   1:L PR[91] 10mm/sec CNT100;
   1:  PR[GP1:91,1] = PR[GP1:90,1] + 73.727;
   1:  PR[GP1:91,2] = PR[GP1:90,2] + 0.302;
   1:L PR[91] 10mm/sec CNT100;
   1:  PR[GP1:91,1] = PR[GP1:90,1] + 73.699;
   1:  PR[GP1:91,2] = PR[GP1:90,2] + 0.551;
   1:L PR[91] 10mm/sec CNT100;
   1:  PR[GP1:91,1] = PR[GP1:90,1] + 71.338;
   1:  PR[GP1:91,2] = PR[GP1:90,2] + 12.899;
   1:L PR[91] 10mm/sec CNT100;
   1:  PR[GP1:91,1] = PR[GP1:90,1] + 64.447;
   1:  PR[GP1:91,2] = PR[GP1:90,2] + 23.769;
   1:L PR[91] 10mm/sec CNT100;
   1:  PR[GP1:91,1] = PR[GP1:90,1] + 64.159;
   1:  PR[GP1:91,2] = PR[GP1:90,2] + 23.993;
   1:L PR[91] 10mm/sec CNT100;
   1:  PR[GP1:91,1] = PR[GP1:90,1] + 54.096;
   1:  PR[GP1:91,2] = PR[GP1:90,2] + 31.348;
   1:L PR[91] 10mm/sec CNT100;
   1:  PR[GP1:91,1] = PR[GP1:90,1] + 52.731;
   1:  PR[GP1:91,2] = PR[GP1:90,2] + 31.773;
   1:L PR[91] 10mm/sec CNT100;
   1:  PR[GP1:91,1] = PR[GP1:90,1] + 41.768;
   1:  PR[GP1:91,2] = PR[GP1:90,2] + 34.681;
   1:L PR[91] 10mm/sec CNT100;
   1:  PR[GP1:91,1] = PR[GP1:90,1] + 38.848;
   1:  PR[GP1:91,2] = PR[GP1:90,2] + 34.517;
   1:L PR[91] 10mm/sec CNT100;
   1:  PR[GP1:91,1] = PR[GP1:90,1] + 29.167;
   1:  PR[GP1:91,2] = PR[GP1:90,2] + 33.430;
   1:L PR[91] 10mm/sec CNT100;
   1:  PR[GP1:91,1] = PR[GP1:90,1] + 24.881;
   1:  PR[GP1:91,2] = PR[GP1:90,2] + 31.548;
   1:L PR[91] 10mm/sec CNT100;
   1:  PR[GP1:91,1] = PR[GP1:90,1] + 17.929;
   1:  PR[GP1:91,2] = PR[GP1:90,2] + 27.897;
   1:L PR[91] 10mm/sec CNT100;
   1:  PR[GP1:91,1] = PR[GP1:90,1] + 13.378;
   1:  PR[GP1:91,2] = PR[GP1:90,2] + 23.438;
   1:L PR[91] 10mm/sec CNT100;
   1:  PR[GP1:91,1] = PR[GP1:90,1] + 9.416;
   1:  PR[GP1:91,2] = PR[GP1:90,2] + 18.841;
   1:L PR[91] 10mm/sec CNT100;
   1:  PR[GP1:91,1] = PR[GP1:90,1] + 6.241;
   1:  PR[GP1:91,2] = PR[GP1:90,2] + 12.001;
   1:L PR[91] 10mm/sec CNT100;
   1:  PR[GP1:91,1] = PR[GP1:90,1] + 4.489;
   1:  PR[GP1:91,2] = PR[GP1:90,2] + 6.941;
   1:L PR[91] 10mm/sec CNT100;
   1:  PR[GP1:91,1] = PR[GP1:90,1] + -5.019;
   1:L PR[91] 10mm/sec CNT100;
   1:  PR[GP1:91,1] = PR[GP1:90,1] + -6.774;
   1:  PR[GP1:91,2] = PR[GP1:90,2] + 12.009;
   1:L PR[91] 10mm/sec CNT100;
   1:  PR[GP1:91,1] = PR[GP1:90,1] + -9.950;
   1:  PR[GP1:91,2] = PR[GP1:90,2] + 18.859;
   1:L PR[91] 10mm/sec CNT100;
   1:  PR[GP1:91,1] = PR[GP1:90,1] + -13.913;
   1:  PR[GP1:91,2] = PR[GP1:90,2] + 23.453;
   1:L PR[91] 10mm/sec CNT100;
   1:  PR[GP1:91,1] = PR[GP1:90,1] + -18.463;
   1:  PR[GP1:91,2] = PR[GP1:90,2] + 27.901;
   1:L PR[91] 10mm/sec CNT100;
   1:  PR[GP1:91,1] = PR[GP1:90,1] + -25.417;
   1:  PR[GP1:91,2] = PR[GP1:90,2] + 31.552;
   1:L PR[91] 10mm/sec CNT100;
   1:  PR[GP1:91,1] = PR[GP1:90,1] + -29.701;
   1:  PR[GP1:91,2] = PR[GP1:90,2] + 33.433;
   1:L PR[91] 10mm/sec CNT100;
   1:  PR[GP1:91,1] = PR[GP1:90,1] + -39.381;
   1:  PR[GP1:91,2] = PR[GP1:90,2] + 34.517;
   1:L PR[91] 10mm/sec CNT100;
   1:  PR[GP1:91,1] = PR[GP1:90,1] + -42.300;
   1:  PR[GP1:91,2] = PR[GP1:90,2] + 34.680;
   1:L PR[91] 10mm/sec CNT100;
   1:  PR[GP1:91,1] = PR[GP1:90,1] + -53.262;
   1:  PR[GP1:91,2] = PR[GP1:90,2] + 31.771;
   1:L PR[91] 10mm/sec CNT100;
   1:  PR[GP1:91,1] = PR[GP1:90,1] + -54.625;
   1:  PR[GP1:91,2] = PR[GP1:90,2] + 31.346;
   1:L PR[91] 10mm/sec CNT100;
   1:  PR[GP1:91,1] = PR[GP1:90,1] + -64.687;
   1:  PR[GP1:91,2] = PR[GP1:90,2] + 23.992;
   1:L PR[91] 10mm/sec CNT100;
   1:  PR[GP1:91,1] = PR[GP1:90,1] + -64.975;
   1:  PR[GP1:91,2] = PR[GP1:90,2] + 23.768;
   1:L PR[91] 10mm/sec CNT100;
   1:  PR[GP1:91,1] = PR[GP1:90,1] + -71.850;
   1:  PR[GP1:91,2] = PR[GP1:90,2] + 12.917;
   1:L PR[91] 10mm/sec CNT100;
   1:  PR[GP1:91,1] = PR[GP1:90,1] + -74.253;
   1:  PR[GP1:91,2] = PR[GP1:90,2] + 0.256;
   1:L PR[91] 10mm/sec CNT100;
   1:  PR[GP1:91,1] = PR[GP1:90,1] + -74.226;
   1:  PR[GP1:91,2] = PR[GP1:90,2] + 0.007;
   1:L PR[91] 10mm/sec CNT100;
   1:  PR[GP1:91,1] = PR[GP1:90,1] + -71.865;
   1:  PR[GP1:91,2] = PR[GP1:90,2] + -12.337;
   1:L PR[91] 10mm/sec CNT100;
   1:  PR[GP1:91,1] = PR[GP1:90,1] + -70.436;
   1:  PR[GP1:91,2] = PR[GP1:90,2] + -14.594;
   1:L PR[91] 10mm/sec CNT100;
   1:  PR[GP1:91,1] = PR[GP1:90,1] + -64.975;
   1:  PR[GP1:91,2] = PR[GP1:90,2] + -23.210;
   1:L PR[91] 10mm/sec CNT100;
   1:  PR[GP1:91,1] = PR[GP1:90,1] + -64.687;
   1:  PR[GP1:91,2] = PR[GP1:90,2] + -23.434;
   1:L PR[91] 10mm/sec CNT100;
   1:  PR[GP1:91,1] = PR[GP1:90,1] + -54.625;
   1:  PR[GP1:91,2] = PR[GP1:90,2] + -30.788;
   1:L PR[91] 10mm/sec CNT100;
   1:  PR[GP1:91,1] = PR[GP1:90,1] + -53.262;
   1:  PR[GP1:91,2] = PR[GP1:90,2] + -31.213;
   1:L PR[91] 10mm/sec CNT100;
   1:  PR[GP1:91,1] = PR[GP1:90,1] + -42.300;
   1:  PR[GP1:91,2] = PR[GP1:90,2] + -34.122;
   1:L PR[91] 10mm/sec CNT100;
   1:  PR[GP1:91,1] = PR[GP1:90,1] + -39.381;
   1:  PR[GP1:91,2] = PR[GP1:90,2] + -33.959;
   1:L PR[91] 10mm/sec CNT100;
   1:  PR[GP1:91,1] = PR[GP1:90,1] + -29.701;
   1:  PR[GP1:91,2] = PR[GP1:90,2] + -32.875;
   1:L PR[91] 10mm/sec CNT100;
   1:  PR[GP1:91,1] = PR[GP1:90,1] + -25.417;
   1:  PR[GP1:91,2] = PR[GP1:90,2] + -30.994;
   1:L PR[91] 10mm/sec CNT100;
   1:  PR[GP1:91,1] = PR[GP1:90,1] + -18.463;
   1:  PR[GP1:91,2] = PR[GP1:90,2] + -27.343;
   1:L PR[91] 10mm/sec CNT100;
   1:  PR[GP1:91,1] = PR[GP1:90,1] + -13.913;
   1:  PR[GP1:91,2] = PR[GP1:90,2] + -22.895;
   1:L PR[91] 10mm/sec CNT100;
   1:  PR[GP1:91,1] = PR[GP1:90,1] + -9.950;
   1:  PR[GP1:91,2] = PR[GP1:90,2] + -18.301;
   1:L PR[91] 10mm/sec CNT100;
   1:  PR[GP1:91,1] = PR[GP1:90,1] + -6.772;
   1:  PR[GP1:91,2] = PR[GP1:90,2] + -11.446;
   1:L PR[91] 10mm/sec CNT100;
   1:  PR[GP1:91,1] = PR[GP1:90,1] + -5.019;
   1:  PR[GP1:91,2] = PR[GP1:90,2] + -6.383;
   1:L PR[91] 10mm/sec CNT100;
   1:  PR[GP1:91,1] = PR[GP1:90,1] + 4.489;
   1:L PR[91] 10mm/sec CNT100;
   1:  PR[GP1:91,1] = PR[GP1:90,1] + 5.797;
   1:  PR[GP1:91,2] = PR[GP1:90,2] + -10.673;
   1:  PR[GP1:91,3] = PR[GP1:90,3] + 20.435;
   1:L PR[91] 10mm/sec CNT100;
   1:  PR[GP1:91,1] = PR[GP1:90,1] + 9.441;
   1:  PR[GP1:91,2] = PR[GP1:90,2] + -18.522;
   1:L PR[91] 10mm/sec CNT100;
   1:  PR[GP1:91,1] = PR[GP1:90,1] + 12.658;
   1:  PR[GP1:91,2] = PR[GP1:90,2] + -22.255;
   1:L PR[91] 10mm/sec CNT100;
   1:  PR[GP1:91,1] = PR[GP1:90,1] + 17.992;
   1:  PR[GP1:91,2] = PR[GP1:90,2] + -27.482;
   1:L PR[91] 10mm/sec CNT100;
   1:  PR[GP1:91,1] = PR[GP1:90,1] + 23.994;
   1:  PR[GP1:91,2] = PR[GP1:90,2] + -30.634;
   1:L PR[91] 10mm/sec CNT100;
   1:  PR[GP1:91,1] = PR[GP1:90,1] + 29.228;
   1:  PR[GP1:91,2] = PR[GP1:90,2] + -32.932;
   1:L PR[91] 10mm/sec CNT100;
   1:  PR[GP1:91,1] = PR[GP1:90,1] + 37.929;
   1:  PR[GP1:91,2] = PR[GP1:90,2] + -33.909;
   1:L PR[91] 10mm/sec CNT100;
   1:  PR[GP1:91,1] = PR[GP1:90,1] + 41.802;
   1:  PR[GP1:91,2] = PR[GP1:90,2] + -34.126;
   1:L PR[91] 10mm/sec CNT100;
   1:  PR[GP1:91,1] = PR[GP1:90,1] + 51.900;
   1:  PR[GP1:91,2] = PR[GP1:90,2] + -31.448;
   1:L PR[91] 10mm/sec CNT100;
   1:  PR[GP1:91,1] = PR[GP1:90,1] + 54.093;
   1:  PR[GP1:91,2] = PR[GP1:90,2] + -30.765;
   1:L PR[91] 10mm/sec CNT100;
   1:  PR[GP1:91,1] = PR[GP1:90,1] + 63.501;
   1:  PR[GP1:91,2] = PR[GP1:90,2] + -23.889;
   1:L PR[91] 10mm/sec CNT100;
   1:  PR[GP1:91,1] = PR[GP1:90,1] + 64.412;
   1:  PR[GP1:91,2] = PR[GP1:90,2] + -23.180;
   1:L PR[91] 10mm/sec CNT100;
   1:  PR[GP1:91,1] = PR[GP1:90,1] + 71.023;
   1:  PR[GP1:91,2] = PR[GP1:90,2] + -12.754;
   1:L PR[91] 10mm/sec CNT100;
   1:  PR[GP1:91,1] = PR[GP1:90,1] + 71.279;
   1:  PR[GP1:91,2] = PR[GP1:90,2] + -12.333;
   1:L PR[91] 10mm/sec CNT100;
   1:  PR[GP1:91,1] = PR[GP1:90,1] + 73.698;
   1:  PR[GP1:91,2] = PR[GP1:90,2] + 0.279;
   1:L PR[91] 10mm/sec CNT100;
   1:  PR[GP1:91,1] = PR[GP1:90,1] + 71.279;
   1:  PR[GP1:91,2] = PR[GP1:90,2] + 12.891;
   1:L PR[91] 10mm/sec CNT100;
   1:  PR[GP1:91,1] = PR[GP1:90,1] + 71.023;
   1:  PR[GP1:91,2] = PR[GP1:90,2] + 13.312;
   1:L PR[91] 10mm/sec CNT100;
   1:  PR[GP1:91,1] = PR[GP1:90,1] + 64.412;
   1:  PR[GP1:91,2] = PR[GP1:90,2] + 23.738;
   1:L PR[91] 10mm/sec CNT100;
   1:  PR[GP1:91,1] = PR[GP1:90,1] + 63.501;
   1:  PR[GP1:91,2] = PR[GP1:90,2] + 24.447;
   1:L PR[91] 10mm/sec CNT100;
   1:  PR[GP1:91,1] = PR[GP1:90,1] + 54.093;
   1:  PR[GP1:91,2] = PR[GP1:90,2] + 31.323;
   1:L PR[91] 10mm/sec CNT100;
   1:  PR[GP1:91,1] = PR[GP1:90,1] + 51.900;
   1:  PR[GP1:91,2] = PR[GP1:90,2] + 32.006;
   1:L PR[91] 10mm/sec CNT100;
   1:  PR[GP1:91,1] = PR[GP1:90,1] + 41.802;
   1:  PR[GP1:91,2] = PR[GP1:90,2] + 34.684;
   1:L PR[91] 10mm/sec CNT100;
   1:  PR[GP1:91,1] = PR[GP1:90,1] + 37.929;
   1:  PR[GP1:91,2] = PR[GP1:90,2] + 34.467;
   1:L PR[91] 10mm/sec CNT100;
   1:  PR[GP1:91,1] = PR[GP1:90,1] + 29.228;
   1:  PR[GP1:91,2] = PR[GP1:90,2] + 33.490;
   1:L PR[91] 10mm/sec CNT100;
   1:  PR[GP1:91,1] = PR[GP1:90,1] + 23.994;
   1:  PR[GP1:91,2] = PR[GP1:90,2] + 31.192;
   1:L PR[91] 10mm/sec CNT100;
   1:  PR[GP1:91,1] = PR[GP1:90,1] + 17.992;
   1:  PR[GP1:91,2] = PR[GP1:90,2] + 28.040;
   1:L PR[91] 10mm/sec CNT100;
   1:  PR[GP1:91,1] = PR[GP1:90,1] + 12.658;
   1:  PR[GP1:91,2] = PR[GP1:90,2] + 22.813;
   1:L PR[91] 10mm/sec CNT100;
   1:  PR[GP1:91,1] = PR[GP1:90,1] + 9.441;
   1:  PR[GP1:91,2] = PR[GP1:90,2] + 19.080;
   1:L PR[91] 10mm/sec CNT100;
   1:  PR[GP1:91,1] = PR[GP1:90,1] + 5.795;
   1:  PR[GP1:91,2] = PR[GP1:90,2] + 11.226;
   1:L PR[91] 10mm/sec CNT100;
   1:  PR[GP1:91,1] = PR[GP1:90,1] + 4.424;
   1:  PR[GP1:91,2] = PR[GP1:90,2] + 7.266;
   1:L PR[91] 10mm/sec CNT100;
   1:  PR[GP1:91,1] = PR[GP1:90,1] + -4.954;
   1:L PR[91] 10mm/sec CNT100;
   1:  PR[GP1:91,1] = PR[GP1:90,1] + -6.328;
   1:  PR[GP1:91,2] = PR[GP1:90,2] + 11.234;
   1:L PR[91] 10mm/sec CNT100;
   1:  PR[GP1:91,1] = PR[GP1:90,1] + -9.975;
   1:  PR[GP1:91,2] = PR[GP1:90,2] + 19.099;
   1:L PR[91] 10mm/sec CNT100;
   1:  PR[GP1:91,1] = PR[GP1:90,1] + -13.193;
   1:  PR[GP1:91,2] = PR[GP1:90,2] + 22.830;
   1:L PR[91] 10mm/sec CNT100;
   1:  PR[GP1:91,1] = PR[GP1:90,1] + -18.527;
   1:  PR[GP1:91,2] = PR[GP1:90,2] + 28.044;
   1:L PR[91] 10mm/sec CNT100;
   1:  PR[GP1:91,1] = PR[GP1:90,1] + -24.530;
   1:  PR[GP1:91,2] = PR[GP1:90,2] + 31.196;
   1:L PR[91] 10mm/sec CNT100;
   1:  PR[GP1:91,1] = PR[GP1:90,1] + -29.762;
   1:  PR[GP1:91,2] = PR[GP1:90,2] + 33.493;
   1:L PR[91] 10mm/sec CNT100;
   1:  PR[GP1:91,1] = PR[GP1:90,1] + -38.463;
   1:  PR[GP1:91,2] = PR[GP1:90,2] + 34.468;
   1:L PR[91] 10mm/sec CNT100;
   1:  PR[GP1:91,1] = PR[GP1:90,1] + -42.334;
   1:  PR[GP1:91,2] = PR[GP1:90,2] + 34.684;
   1:L PR[91] 10mm/sec CNT100;
   1:  PR[GP1:91,1] = PR[GP1:90,1] + -52.432;
   1:  PR[GP1:91,2] = PR[GP1:90,2] + 32.004;
   1:L PR[91] 10mm/sec CNT100;
   1:  PR[GP1:91,1] = PR[GP1:90,1] + -54.623;
   1:  PR[GP1:91,2] = PR[GP1:90,2] + 31.321;
   1:L PR[91] 10mm/sec CNT100;
   1:  PR[GP1:91,1] = PR[GP1:90,1] + -64.030;
   1:  PR[GP1:91,2] = PR[GP1:90,2] + 24.446;
   1:L PR[91] 10mm/sec CNT100;
   1:  PR[GP1:91,1] = PR[GP1:90,1] + -64.940;
   1:  PR[GP1:91,2] = PR[GP1:90,2] + 23.737;
   1:L PR[91] 10mm/sec CNT100;
   1:  PR[GP1:91,1] = PR[GP1:90,1] + -71.550;
   1:  PR[GP1:91,2] = PR[GP1:90,2] + 13.309;
   1:L PR[91] 10mm/sec CNT100;
   1:  PR[GP1:91,1] = PR[GP1:90,1] + -71.806;
   1:  PR[GP1:91,2] = PR[GP1:90,2] + 12.888;
   1:L PR[91] 10mm/sec CNT100;
   1:  PR[GP1:91,1] = PR[GP1:90,1] + -74.224;
   1:  PR[GP1:91,2] = PR[GP1:90,2] + 0.279;
   1:L PR[91] 10mm/sec CNT100;
   1:  PR[GP1:91,1] = PR[GP1:90,1] + -71.806;
   1:  PR[GP1:91,2] = PR[GP1:90,2] + -12.329;
   1:L PR[91] 10mm/sec CNT100;
   1:  PR[GP1:91,1] = PR[GP1:90,1] + -71.550;
   1:  PR[GP1:91,2] = PR[GP1:90,2] + -12.751;
   1:L PR[91] 10mm/sec CNT100;
   1:  PR[GP1:91,1] = PR[GP1:90,1] + -64.940;
   1:  PR[GP1:91,2] = PR[GP1:90,2] + -23.179;
   1:L PR[91] 10mm/sec CNT100;
   1:  PR[GP1:91,1] = PR[GP1:90,1] + -64.030;
   1:  PR[GP1:91,2] = PR[GP1:90,2] + -23.888;
   1:L PR[91] 10mm/sec CNT100;
   1:  PR[GP1:91,1] = PR[GP1:90,1] + -54.623;
   1:  PR[GP1:91,2] = PR[GP1:90,2] + -30.763;
   1:L PR[91] 10mm/sec CNT100;
   1:  PR[GP1:91,1] = PR[GP1:90,1] + -52.432;
   1:  PR[GP1:91,2] = PR[GP1:90,2] + -31.446;
   1:L PR[91] 10mm/sec CNT100;
   1:  PR[GP1:91,1] = PR[GP1:90,1] + -42.334;
   1:  PR[GP1:91,2] = PR[GP1:90,2] + -34.126;
   1:L PR[91] 10mm/sec CNT100;
   1:  PR[GP1:91,1] = PR[GP1:90,1] + -38.463;
   1:  PR[GP1:91,2] = PR[GP1:90,2] + -33.910;
   1:L PR[91] 10mm/sec CNT100;
   1:  PR[GP1:91,1] = PR[GP1:90,1] + -29.762;
   1:  PR[GP1:91,2] = PR[GP1:90,2] + -32.935;
   1:L PR[91] 10mm/sec CNT100;
   1:  PR[GP1:91,1] = PR[GP1:90,1] + -24.530;
   1:  PR[GP1:91,2] = PR[GP1:90,2] + -30.638;
   1:L PR[91] 10mm/sec CNT100;
   1:  PR[GP1:91,1] = PR[GP1:90,1] + -18.527;
   1:  PR[GP1:91,2] = PR[GP1:90,2] + -27.486;
   1:L PR[91] 10mm/sec CNT100;
   1:  PR[GP1:91,1] = PR[GP1:90,1] + -13.193;
   1:  PR[GP1:91,2] = PR[GP1:90,2] + -22.272;
   1:L PR[91] 10mm/sec CNT100;
   1:  PR[GP1:91,1] = PR[GP1:90,1] + -9.975;
   1:  PR[GP1:91,2] = PR[GP1:90,2] + -18.541;
   1:L PR[91] 10mm/sec CNT100;
   1:  PR[GP1:91,1] = PR[GP1:90,1] + -6.326;
   1:  PR[GP1:91,2] = PR[GP1:90,2] + -10.671;
   1:L PR[91] 10mm/sec CNT100;
   1:  PR[GP1:91,1] = PR[GP1:90,1] + -4.954;
   1:  PR[GP1:91,2] = PR[GP1:90,2] + -6.708;
   1:L PR[91] 10mm/sec CNT100;
   1:  PR[GP1:91,1] = PR[GP1:90,1] + 4.424;
   1:L PR[91] 10mm/sec CNT100;
   1:  PR[GP1:91,1] = PR[GP1:90,1] + 5.351;
   1:  PR[GP1:91,2] = PR[GP1:90,2] + -9.899;
   1:  PR[GP1:91,3] = PR[GP1:90,3] + 21.045;
   1:L PR[91] 10mm/sec CNT100;
   1:  PR[GP1:91,1] = PR[GP1:90,1] + 9.465;
   1:  PR[GP1:91,2] = PR[GP1:90,2] + -18.761;
   1:L PR[91] 10mm/sec CNT100;
   1:  PR[GP1:91,1] = PR[GP1:90,1] + 11.938;
   1:  PR[GP1:91,2] = PR[GP1:90,2] + -21.630;
   1:L PR[91] 10mm/sec CNT100;
   1:  PR[GP1:91,1] = PR[GP1:90,1] + 18.056;
   1:  PR[GP1:91,2] = PR[GP1:90,2] + -27.625;
   1:L PR[91] 10mm/sec CNT100;
   1:  PR[GP1:91,1] = PR[GP1:90,1] + 23.107;
   1:  PR[GP1:91,2] = PR[GP1:90,2] + -30.278;
   1:L PR[91] 10mm/sec CNT100;
   1:  PR[GP1:91,1] = PR[GP1:90,1] + 29.289;
   1:  PR[GP1:91,2] = PR[GP1:90,2] + -32.992;
   1:L PR[91] 10mm/sec CNT100;
   1:  PR[GP1:91,1] = PR[GP1:90,1] + 37.011;
   1:  PR[GP1:91,2] = PR[GP1:90,2] + -33.859;
   1:L PR[91] 10mm/sec CNT100;
   1:  PR[GP1:91,1] = PR[GP1:90,1] + 41.836;
   1:  PR[GP1:91,2] = PR[GP1:90,2] + -34.130;
   1:L PR[91] 10mm/sec CNT100;
   1:  PR[GP1:91,1] = PR[GP1:90,1] + 51.070;
   1:  PR[GP1:91,2] = PR[GP1:90,2] + -31.680;
   1:L PR[91] 10mm/sec CNT100;
   1:  PR[GP1:91,1] = PR[GP1:90,1] + 54.091;
   1:  PR[GP1:91,2] = PR[GP1:90,2] + -30.740;
   1:L PR[91] 10mm/sec CNT100;
   1:  PR[GP1:91,1] = PR[GP1:90,1] + 62.844;
   1:  PR[GP1:91,2] = PR[GP1:90,2] + -24.343;
   1:L PR[91] 10mm/sec CNT100;
   1:  PR[GP1:91,1] = PR[GP1:90,1] + 64.377;
   1:  PR[GP1:91,2] = PR[GP1:90,2] + -23.150;
   1:L PR[91] 10mm/sec CNT100;
   1:  PR[GP1:91,1] = PR[GP1:90,1] + 70.589;
   1:  PR[GP1:91,2] = PR[GP1:90,2] + -13.354;
   1:L PR[91] 10mm/sec CNT100;
   1:  PR[GP1:91,1] = PR[GP1:90,1] + 71.221;
   1:  PR[GP1:91,2] = PR[GP1:90,2] + -12.314;
   1:L PR[91] 10mm/sec CNT100;
   1:  PR[GP1:91,1] = PR[GP1:90,1] + 73.632;
   1:  PR[GP1:91,2] = PR[GP1:90,2] + 0.279;
   1:L PR[91] 10mm/sec CNT100;
   1:  PR[GP1:91,1] = PR[GP1:90,1] + 71.221;
   1:  PR[GP1:91,2] = PR[GP1:90,2] + 12.872;
   1:L PR[91] 10mm/sec CNT100;
   1:  PR[GP1:91,1] = PR[GP1:90,1] + 70.589;
   1:  PR[GP1:91,2] = PR[GP1:90,2] + 13.912;
   1:L PR[91] 10mm/sec CNT100;
   1:  PR[GP1:91,1] = PR[GP1:90,1] + 64.377;
   1:  PR[GP1:91,2] = PR[GP1:90,2] + 23.708;
   1:L PR[91] 10mm/sec CNT100;
   1:  PR[GP1:91,1] = PR[GP1:90,1] + 62.844;
   1:  PR[GP1:91,2] = PR[GP1:90,2] + 24.901;
   1:L PR[91] 10mm/sec CNT100;
   1:  PR[GP1:91,1] = PR[GP1:90,1] + 54.091;
   1:  PR[GP1:91,2] = PR[GP1:90,2] + 31.298;
   1:L PR[91] 10mm/sec CNT100;
   1:  PR[GP1:91,1] = PR[GP1:90,1] + 51.070;
   1:  PR[GP1:91,2] = PR[GP1:90,2] + 32.239;
   1:L PR[91] 10mm/sec CNT100;
   1:  PR[GP1:91,1] = PR[GP1:90,1] + 41.836;
   1:  PR[GP1:91,2] = PR[GP1:90,2] + 34.688;
   1:L PR[91] 10mm/sec CNT100;
   1:  PR[GP1:91,1] = PR[GP1:90,1] + 37.011;
   1:  PR[GP1:91,2] = PR[GP1:90,2] + 34.417;
   1:L PR[91] 10mm/sec CNT100;
   1:  PR[GP1:91,1] = PR[GP1:90,1] + 29.289;
   1:  PR[GP1:91,2] = PR[GP1:90,2] + 33.550;
   1:L PR[91] 10mm/sec CNT100;
   1:  PR[GP1:91,1] = PR[GP1:90,1] + 23.107;
   1:  PR[GP1:91,2] = PR[GP1:90,2] + 30.836;
   1:L PR[91] 10mm/sec CNT100;
   1:  PR[GP1:91,1] = PR[GP1:90,1] + 18.056;
   1:  PR[GP1:91,2] = PR[GP1:90,2] + 28.183;
   1:L PR[91] 10mm/sec CNT100;
   1:  PR[GP1:91,1] = PR[GP1:90,1] + 11.938;
   1:  PR[GP1:91,2] = PR[GP1:90,2] + 22.188;
   1:L PR[91] 10mm/sec CNT100;
   1:  PR[GP1:91,1] = PR[GP1:90,1] + 9.465;
   1:  PR[GP1:91,2] = PR[GP1:90,2] + 19.319;
   1:L PR[91] 10mm/sec CNT100;
   1:  PR[GP1:91,1] = PR[GP1:90,1] + 5.349;
   1:  PR[GP1:91,2] = PR[GP1:90,2] + 10.451;
   1:L PR[91] 10mm/sec CNT100;
   1:  PR[GP1:91,1] = PR[GP1:90,1] + 4.359;
   1:  PR[GP1:91,2] = PR[GP1:90,2] + 7.591;
   1:L PR[91] 10mm/sec CNT100;
   1:  PR[GP1:91,1] = PR[GP1:90,1] + -4.889;
   1:L PR[91] 10mm/sec CNT100;
   1:  PR[GP1:91,1] = PR[GP1:90,1] + -5.882;
   1:  PR[GP1:91,2] = PR[GP1:90,2] + 10.460;
   1:L PR[91] 10mm/sec CNT100;
   1:  PR[GP1:91,1] = PR[GP1:90,1] + -10.000;
   1:  PR[GP1:91,2] = PR[GP1:90,2] + 19.339;
   1:L PR[91] 10mm/sec CNT100;
   1:  PR[GP1:91,1] = PR[GP1:90,1] + -12.474;
   1:  PR[GP1:91,2] = PR[GP1:90,2] + 22.207;
   1:L PR[91] 10mm/sec CNT100;
   1:  PR[GP1:91,1] = PR[GP1:90,1] + -18.591;
   1:  PR[GP1:91,2] = PR[GP1:90,2] + 28.187;
   1:L PR[91] 10mm/sec CNT100;
   1:  PR[GP1:91,1] = PR[GP1:90,1] + -23.644;
   1:  PR[GP1:91,2] = PR[GP1:90,2] + 30.840;
   1:L PR[91] 10mm/sec CNT100;
   1:  PR[GP1:91,1] = PR[GP1:90,1] + -29.824;
   1:  PR[GP1:91,2] = PR[GP1:90,2] + 33.553;
   1:L PR[91] 10mm/sec CNT100;
   1:  PR[GP1:91,1] = PR[GP1:90,1] + -37.546;
   1:  PR[GP1:91,2] = PR[GP1:90,2] + 34.418;
   1:L PR[91] 10mm/sec CNT100;
   1:  PR[GP1:91,1] = PR[GP1:90,1] + -42.368;
   1:  PR[GP1:91,2] = PR[GP1:90,2] + 34.687;
   1:L PR[91] 10mm/sec CNT100;
   1:  PR[GP1:91,1] = PR[GP1:90,1] + -51.602;
   1:  PR[GP1:91,2] = PR[GP1:90,2] + 32.237;
   1:L PR[91] 10mm/sec CNT100;
   1:  PR[GP1:91,1] = PR[GP1:90,1] + -54.621;
   1:  PR[GP1:91,2] = PR[GP1:90,2] + 31.296;
   1:L PR[91] 10mm/sec CNT100;
   1:  PR[GP1:91,1] = PR[GP1:90,1] + -63.373;
   1:  PR[GP1:91,2] = PR[GP1:90,2] + 24.899;
   1:L PR[91] 10mm/sec CNT100;
   1:  PR[GP1:91,1] = PR[GP1:90,1] + -64.905;
   1:  PR[GP1:91,2] = PR[GP1:90,2] + 23.707;
   1:L PR[91] 10mm/sec CNT100;
   1:  PR[GP1:91,1] = PR[GP1:90,1] + -71.116;
   1:  PR[GP1:91,2] = PR[GP1:90,2] + 13.908;
   1:L PR[91] 10mm/sec CNT100;
   1:  PR[GP1:91,1] = PR[GP1:90,1] + -71.748;
   1:  PR[GP1:91,2] = PR[GP1:90,2] + 12.868;
   1:L PR[91] 10mm/sec CNT100;
   1:  PR[GP1:91,1] = PR[GP1:90,1] + -74.158;
   1:  PR[GP1:91,2] = PR[GP1:90,2] + 0.279;
   1:L PR[91] 10mm/sec CNT100;
   1:  PR[GP1:91,1] = PR[GP1:90,1] + -71.748;
   1:  PR[GP1:91,2] = PR[GP1:90,2] + -12.310;
   1:L PR[91] 10mm/sec CNT100;
   1:  PR[GP1:91,1] = PR[GP1:90,1] + -71.115;
   1:  PR[GP1:91,2] = PR[GP1:90,2] + -13.350;
   1:L PR[91] 10mm/sec CNT100;
   1:  PR[GP1:91,1] = PR[GP1:90,1] + -64.905;
   1:  PR[GP1:91,2] = PR[GP1:90,2] + -23.149;
   1:L PR[91] 10mm/sec CNT100;
   1:  PR[GP1:91,1] = PR[GP1:90,1] + -63.373;
   1:  PR[GP1:91,2] = PR[GP1:90,2] + -24.341;
   1:L PR[91] 10mm/sec CNT100;
   1:  PR[GP1:91,1] = PR[GP1:90,1] + -54.621;
   1:  PR[GP1:91,2] = PR[GP1:90,2] + -30.738;
   1:L PR[91] 10mm/sec CNT100;
   1:  PR[GP1:91,1] = PR[GP1:90,1] + -51.602;
   1:  PR[GP1:91,2] = PR[GP1:90,2] + -31.679;
   1:L PR[91] 10mm/sec CNT100;
   1:  PR[GP1:91,1] = PR[GP1:90,1] + -42.368;
   1:  PR[GP1:91,2] = PR[GP1:90,2] + -34.129;
   1:L PR[91] 10mm/sec CNT100;
   1:  PR[GP1:91,1] = PR[GP1:90,1] + -37.545;
   1:  PR[GP1:91,2] = PR[GP1:90,2] + -33.860;
   1:L PR[91] 10mm/sec CNT100;
   1:  PR[GP1:91,1] = PR[GP1:90,1] + -29.824;
   1:  PR[GP1:91,2] = PR[GP1:90,2] + -32.995;
   1:L PR[91] 10mm/sec CNT100;
   1:  PR[GP1:91,1] = PR[GP1:90,1] + -23.644;
   1:  PR[GP1:91,2] = PR[GP1:90,2] + -30.282;
   1:L PR[91] 10mm/sec CNT100;
   1:  PR[GP1:91,1] = PR[GP1:90,1] + -18.591;
   1:  PR[GP1:91,2] = PR[GP1:90,2] + -27.629;
   1:L PR[91] 10mm/sec CNT100;
   1:  PR[GP1:91,1] = PR[GP1:90,1] + -12.474;
   1:  PR[GP1:91,2] = PR[GP1:90,2] + -21.649;
   1:L PR[91] 10mm/sec CNT100;
   1:  PR[GP1:91,1] = PR[GP1:90,1] + -10.000;
   1:  PR[GP1:91,2] = PR[GP1:90,2] + -18.781;
   1:L PR[91] 10mm/sec CNT100;
   1:  PR[GP1:91,1] = PR[GP1:90,1] + -5.880;
   1:  PR[GP1:91,2] = PR[GP1:90,2] + -9.896;
   1:L PR[91] 10mm/sec CNT100;
   1:  PR[GP1:91,1] = PR[GP1:90,1] + -4.889;
   1:  PR[GP1:91,2] = PR[GP1:90,2] + -7.033;
   1:L PR[91] 10mm/sec CNT100;
   1:  PR[GP1:91,1] = PR[GP1:90,1] + 4.359;
   1:L PR[91] 10mm/sec CNT100;
   1:  PR[GP1:91,1] = PR[GP1:90,1] + 4.905;
   1:  PR[GP1:91,2] = PR[GP1:90,2] + -9.125;
   1:  PR[GP1:91,3] = PR[GP1:90,3] + 21.655;
   1:L PR[91] 10mm/sec CNT100;
   1:  PR[GP1:91,1] = PR[GP1:90,1] + 9.489;
   1:  PR[GP1:91,2] = PR[GP1:90,2] + -18.999;
   1:L PR[91] 10mm/sec CNT100;
   1:  PR[GP1:91,1] = PR[GP1:90,1] + 11.218;
   1:  PR[GP1:91,2] = PR[GP1:90,2] + -21.005;
   1:L PR[91] 10mm/sec CNT100;
   1:  PR[GP1:91,1] = PR[GP1:90,1] + 18.119;
   1:  PR[GP1:91,2] = PR[GP1:90,2] + -27.768;
   1:L PR[91] 10mm/sec CNT100;
   1:  PR[GP1:91,1] = PR[GP1:90,1] + 22.220;
   1:  PR[GP1:91,2] = PR[GP1:90,2] + -29.921;
   1:L PR[91] 10mm/sec CNT100;
   1:  PR[GP1:91,1] = PR[GP1:90,1] + 29.350;
   1:  PR[GP1:91,2] = PR[GP1:90,2] + -33.052;
   1:L PR[91] 10mm/sec CNT100;
   1:  PR[GP1:91,1] = PR[GP1:90,1] + 36.092;
   1:  PR[GP1:91,2] = PR[GP1:90,2] + -33.809;
   1:L PR[91] 10mm/sec CNT100;
   1:  PR[GP1:91,1] = PR[GP1:90,1] + 41.870;
   1:  PR[GP1:91,2] = PR[GP1:90,2] + -34.133;
   1:L PR[91] 10mm/sec CNT100;
   1:  PR[GP1:91,1] = PR[GP1:90,1] + 50.239;
   1:  PR[GP1:91,2] = PR[GP1:90,2] + -31.913;
   1:L PR[91] 10mm/sec CNT100;
   1:  PR[GP1:91,1] = PR[GP1:90,1] + 54.089;
   1:  PR[GP1:91,2] = PR[GP1:90,2] + -30.715;
   1:L PR[91] 10mm/sec CNT100;
   1:  PR[GP1:91,1] = PR[GP1:90,1] + 62.186;
   1:  PR[GP1:91,2] = PR[GP1:90,2] + -24.797;
   1:L PR[91] 10mm/sec CNT100;
   1:  PR[GP1:91,1] = PR[GP1:90,1] + 64.342;
   1:  PR[GP1:91,2] = PR[GP1:90,2] + -23.120;
   1:L PR[91] 10mm/sec CNT100;
   1:  PR[GP1:91,1] = PR[GP1:90,1] + 70.154;
   1:  PR[GP1:91,2] = PR[GP1:90,2] + -13.953;
   1:L PR[91] 10mm/sec CNT100;
   1:  PR[GP1:91,1] = PR[GP1:90,1] + 71.164;
   1:  PR[GP1:91,2] = PR[GP1:90,2] + -12.295;
   1:L PR[91] 10mm/sec CNT100;
   1:  PR[GP1:91,1] = PR[GP1:90,1] + 73.565;
   1:  PR[GP1:91,2] = PR[GP1:90,2] + 0.279;
   1:L PR[91] 10mm/sec CNT100;
   1:  PR[GP1:91,1] = PR[GP1:90,1] + 71.476;
   1:  PR[GP1:91,2] = PR[GP1:90,2] + 11.155;
   1:L PR[91] 10mm/sec CNT100;
   1:  PR[GP1:91,1] = PR[GP1:90,1] + 71.163;
   1:  PR[GP1:91,2] = PR[GP1:90,2] + 12.855;
   1:L PR[91] 10mm/sec CNT100;
   1:  PR[GP1:91,1] = PR[GP1:90,1] + 70.154;
   1:  PR[GP1:91,2] = PR[GP1:90,2] + 14.511;
   1:L PR[91] 10mm/sec CNT100;
   1:  PR[GP1:91,1] = PR[GP1:90,1] + 64.342;
   1:  PR[GP1:91,2] = PR[GP1:90,2] + 23.678;
   1:L PR[91] 10mm/sec CNT100;
   1:  PR[GP1:91,1] = PR[GP1:90,1] + 62.187;
   1:  PR[GP1:91,2] = PR[GP1:90,2] + 25.355;
   1:L PR[91] 10mm/sec CNT100;
   1:  PR[GP1:91,1] = PR[GP1:90,1] + 54.089;
   1:  PR[GP1:91,2] = PR[GP1:90,2] + 31.273;
   1:L PR[91] 10mm/sec CNT100;
   1:  PR[GP1:91,1] = PR[GP1:90,1] + 50.239;
   1:  PR[GP1:91,2] = PR[GP1:90,2] + 32.471;
   1:L PR[91] 10mm/sec CNT100;
   1:  PR[GP1:91,1] = PR[GP1:90,1] + 41.870;
   1:  PR[GP1:91,2] = PR[GP1:90,2] + 34.691;
   1:L PR[91] 10mm/sec CNT100;
   1:  PR[GP1:91,1] = PR[GP1:90,1] + 36.092;
   1:  PR[GP1:91,2] = PR[GP1:90,2] + 34.367;
   1:L PR[91] 10mm/sec CNT100;
   1:  PR[GP1:91,1] = PR[GP1:90,1] + 29.350;
   1:  PR[GP1:91,2] = PR[GP1:90,2] + 33.610;
   1:L PR[91] 10mm/sec CNT100;
   1:  PR[GP1:91,1] = PR[GP1:90,1] + 22.220;
   1:  PR[GP1:91,2] = PR[GP1:90,2] + 30.479;
   1:L PR[91] 10mm/sec CNT100;
   1:  PR[GP1:91,1] = PR[GP1:90,1] + 18.119;
   1:  PR[GP1:91,2] = PR[GP1:90,2] + 28.326;
   1:L PR[91] 10mm/sec CNT100;
   1:  PR[GP1:91,1] = PR[GP1:90,1] + 11.218;
   1:  PR[GP1:91,2] = PR[GP1:90,2] + 21.563;
   1:L PR[91] 10mm/sec CNT100;
   1:  PR[GP1:91,1] = PR[GP1:90,1] + 9.489;
   1:  PR[GP1:91,2] = PR[GP1:90,2] + 19.557;
   1:L PR[91] 10mm/sec CNT100;
   1:  PR[GP1:91,1] = PR[GP1:90,1] + 4.903;
   1:  PR[GP1:91,2] = PR[GP1:90,2] + 9.677;
   1:L PR[91] 10mm/sec CNT100;
   1:  PR[GP1:91,1] = PR[GP1:90,1] + 4.293;
   1:  PR[GP1:91,2] = PR[GP1:90,2] + 7.916;
   1:L PR[91] 10mm/sec CNT100;
   1:  PR[GP1:91,1] = PR[GP1:90,1] + -4.824;
   1:L PR[91] 10mm/sec CNT100;
   1:  PR[GP1:91,1] = PR[GP1:90,1] + -5.436;
   1:  PR[GP1:91,2] = PR[GP1:90,2] + 9.685;
   1:L PR[91] 10mm/sec CNT100;
   1:  PR[GP1:91,1] = PR[GP1:90,1] + -10.024;
   1:  PR[GP1:91,2] = PR[GP1:90,2] + 19.579;
   1:L PR[91] 10mm/sec CNT100;
   1:  PR[GP1:91,1] = PR[GP1:90,1] + -11.754;
   1:  PR[GP1:91,2] = PR[GP1:90,2] + 21.585;
   1:L PR[91] 10mm/sec CNT100;
   1:  PR[GP1:91,1] = PR[GP1:90,1] + -18.655;
   1:  PR[GP1:91,2] = PR[GP1:90,2] + 28.330;
   1:L PR[91] 10mm/sec CNT100;
   1:  PR[GP1:91,1] = PR[GP1:90,1] + -22.758;
   1:  PR[GP1:91,2] = PR[GP1:90,2] + 30.484;
   1:L PR[91] 10mm/sec CNT100;
   1:  PR[GP1:91,1] = PR[GP1:90,1] + -29.885;
   1:  PR[GP1:91,2] = PR[GP1:90,2] + 33.613;
   1:L PR[91] 10mm/sec CNT100;
   1:  PR[GP1:91,1] = PR[GP1:90,1] + -36.628;
   1:  PR[GP1:91,2] = PR[GP1:90,2] + 34.369;
   1:L PR[91] 10mm/sec CNT100;
   1:  PR[GP1:91,1] = PR[GP1:90,1] + -42.403;
   1:  PR[GP1:91,2] = PR[GP1:90,2] + 34.691;
   1:L PR[91] 10mm/sec CNT100;
   1:  PR[GP1:91,1] = PR[GP1:90,1] + -50.772;
   1:  PR[GP1:91,2] = PR[GP1:90,2] + 32.470;
   1:L PR[91] 10mm/sec CNT100;
   1:  PR[GP1:91,1] = PR[GP1:90,1] + -54.619;
   1:  PR[GP1:91,2] = PR[GP1:90,2] + 31.271;
   1:L PR[91] 10mm/sec CNT100;
   1:  PR[GP1:91,1] = PR[GP1:90,1] + -62.716;
   1:  PR[GP1:91,2] = PR[GP1:90,2] + 25.353;
   1:L PR[91] 10mm/sec CNT100;
   1:  PR[GP1:91,1] = PR[GP1:90,1] + -64.870;
   1:  PR[GP1:91,2] = PR[GP1:90,2] + 23.677;
   1:L PR[91] 10mm/sec CNT100;
   1:  PR[GP1:91,1] = PR[GP1:90,1] + -70.681;
   1:  PR[GP1:91,2] = PR[GP1:90,2] + 14.508;
   1:L PR[91] 10mm/sec CNT100;
   1:  PR[GP1:91,1] = PR[GP1:90,1] + -71.690;
   1:  PR[GP1:91,2] = PR[GP1:90,2] + 12.848;
   1:L PR[91] 10mm/sec CNT100;
   1:  PR[GP1:91,1] = PR[GP1:90,1] + -74.091;
   1:  PR[GP1:91,2] = PR[GP1:90,2] + 0.279;
   1:L PR[91] 10mm/sec CNT100;
   1:  PR[GP1:91,1] = PR[GP1:90,1] + -72.003;
   1:  PR[GP1:91,2] = PR[GP1:90,2] + -10.593;
   1:L PR[91] 10mm/sec CNT100;
   1:  PR[GP1:91,1] = PR[GP1:90,1] + -71.689;
   1:  PR[GP1:91,2] = PR[GP1:90,2] + -12.292;
   1:L PR[91] 10mm/sec CNT100;
   1:  PR[GP1:91,1] = PR[GP1:90,1] + -70.681;
   1:  PR[GP1:91,2] = PR[GP1:90,2] + -13.950;
   1:L PR[91] 10mm/sec CNT100;
   1:  PR[GP1:91,1] = PR[GP1:90,1] + -64.870;
   1:  PR[GP1:91,2] = PR[GP1:90,2] + -23.119;
   1:L PR[91] 10mm/sec CNT100;
   1:  PR[GP1:91,1] = PR[GP1:90,1] + -62.716;
   1:  PR[GP1:91,2] = PR[GP1:90,2] + -24.795;
   1:L PR[91] 10mm/sec CNT100;
   1:  PR[GP1:91,1] = PR[GP1:90,1] + -54.619;
   1:  PR[GP1:91,2] = PR[GP1:90,2] + -30.713;
   1:L PR[91] 10mm/sec CNT100;
   1:  PR[GP1:91,1] = PR[GP1:90,1] + -50.772;
   1:  PR[GP1:91,2] = PR[GP1:90,2] + -31.912;
   1:L PR[91] 10mm/sec CNT100;
   1:  PR[GP1:91,1] = PR[GP1:90,1] + -42.403;
   1:  PR[GP1:91,2] = PR[GP1:90,2] + -34.133;
   1:L PR[91] 10mm/sec CNT100;
   1:  PR[GP1:91,1] = PR[GP1:90,1] + -36.627;
   1:  PR[GP1:91,2] = PR[GP1:90,2] + -33.810;
   1:L PR[91] 10mm/sec CNT100;
   1:  PR[GP1:91,1] = PR[GP1:90,1] + -29.885;
   1:  PR[GP1:91,2] = PR[GP1:90,2] + -33.055;
   1:L PR[91] 10mm/sec CNT100;
   1:  PR[GP1:91,1] = PR[GP1:90,1] + -22.758;
   1:  PR[GP1:91,2] = PR[GP1:90,2] + -29.926;
   1:L PR[91] 10mm/sec CNT100;
   1:  PR[GP1:91,1] = PR[GP1:90,1] + -18.655;
   1:  PR[GP1:91,2] = PR[GP1:90,2] + -27.772;
   1:L PR[91] 10mm/sec CNT100;
   1:  PR[GP1:91,1] = PR[GP1:90,1] + -11.754;
   1:  PR[GP1:91,2] = PR[GP1:90,2] + -21.026;
   1:L PR[91] 10mm/sec CNT100;
   1:  PR[GP1:91,1] = PR[GP1:90,1] + -10.024;
   1:  PR[GP1:91,2] = PR[GP1:90,2] + -19.021;
   1:L PR[91] 10mm/sec CNT100;
   1:  PR[GP1:91,1] = PR[GP1:90,1] + -5.434;
   1:  PR[GP1:91,2] = PR[GP1:90,2] + -9.120;
   1:L PR[91] 10mm/sec CNT100;
   1:  PR[GP1:91,1] = PR[GP1:90,1] + -4.824;
   1:  PR[GP1:91,2] = PR[GP1:90,2] + -7.358;
   1:L PR[91] 10mm/sec CNT100;
   1:  PR[GP1:91,1] = PR[GP1:90,1] + 4.293;
   1:L PR[91] 10mm/sec CNT100;
   1:  PR[GP1:91,1] = PR[GP1:90,1] + 4.459;
   1:  PR[GP1:91,2] = PR[GP1:90,2] + -8.352;
   1:  PR[GP1:91,3] = PR[GP1:90,3] + 22.265;
   1:L PR[91] 10mm/sec CNT100;
   1:  PR[GP1:91,1] = PR[GP1:90,1] + 9.513;
   1:  PR[GP1:91,2] = PR[GP1:90,2] + -19.238;
   1:L PR[91] 10mm/sec CNT100;
   1:  PR[GP1:91,1] = PR[GP1:90,1] + 10.498;
   1:  PR[GP1:91,2] = PR[GP1:90,2] + -20.380;
   1:L PR[91] 10mm/sec CNT100;
   1:  PR[GP1:91,1] = PR[GP1:90,1] + 18.182;
   1:  PR[GP1:91,2] = PR[GP1:90,2] + -27.911;
   1:L PR[91] 10mm/sec CNT100;
   1:  PR[GP1:91,1] = PR[GP1:90,1] + 21.333;
   1:  PR[GP1:91,2] = PR[GP1:90,2] + -29.565;
   1:L PR[91] 10mm/sec CNT100;
   1:  PR[GP1:91,1] = PR[GP1:90,1] + 29.411;
   1:  PR[GP1:91,2] = PR[GP1:90,2] + -33.112;
   1:L PR[91] 10mm/sec CNT100;
   1:  PR[GP1:91,1] = PR[GP1:90,1] + 35.173;
   1:  PR[GP1:91,2] = PR[GP1:90,2] + -33.759;
   1:L PR[91] 10mm/sec CNT100;
   1:  PR[GP1:91,1] = PR[GP1:90,1] + 41.904;
   1:  PR[GP1:91,2] = PR[GP1:90,2] + -34.137;
   1:L PR[91] 10mm/sec CNT100;
   1:  PR[GP1:91,1] = PR[GP1:90,1] + 49.409;
   1:  PR[GP1:91,2] = PR[GP1:90,2] + -32.146;
   1:L PR[91] 10mm/sec CNT100;
   1:  PR[GP1:91,1] = PR[GP1:90,1] + 54.087;
   1:  PR[GP1:91,2] = PR[GP1:90,2] + -30.690;
   1:L PR[91] 10mm/sec CNT100;
   1:  PR[GP1:91,1] = PR[GP1:90,1] + 61.529;
   1:  PR[GP1:91,2] = PR[GP1:90,2] + -25.250;
   1:L PR[91] 10mm/sec CNT100;
   1:  PR[GP1:91,1] = PR[GP1:90,1] + 64.306;
   1:  PR[GP1:91,2] = PR[GP1:90,2] + -23.090;
   1:L PR[91] 10mm/sec CNT100;
   1:  PR[GP1:91,1] = PR[GP1:90,1] + 69.719;
   1:  PR[GP1:91,2] = PR[GP1:90,2] + -14.553;
   1:L PR[91] 10mm/sec CNT100;
   1:  PR[GP1:91,1] = PR[GP1:90,1] + 71.106;
   1:  PR[GP1:91,2] = PR[GP1:90,2] + -12.275;
   1:L PR[91] 10mm/sec CNT100;
   1:  PR[GP1:91,1] = PR[GP1:90,1] + 73.132;
   1:  PR[GP1:91,2] = PR[GP1:90,2] + -1.711;
   1:L PR[91] 10mm/sec CNT100;
   1:  PR[GP1:91,1] = PR[GP1:90,1] + 73.499;
   1:  PR[GP1:91,2] = PR[GP1:90,2] + 0.277;
   1:L PR[91] 10mm/sec CNT100;
   1:  PR[GP1:91,1] = PR[GP1:90,1] + 71.536;
   1:  PR[GP1:91,2] = PR[GP1:90,2] + 10.498;
   1:L PR[91] 10mm/sec CNT100;
   1:  PR[GP1:91,1] = PR[GP1:90,1] + 71.105;
   1:  PR[GP1:91,2] = PR[GP1:90,2] + 12.835;
   1:L PR[91] 10mm/sec CNT100;
   1:  PR[GP1:91,1] = PR[GP1:90,1] + 69.719;
   1:  PR[GP1:91,2] = PR[GP1:90,2] + 15.111;
   1:L PR[91] 10mm/sec CNT100;
   1:  PR[GP1:91,1] = PR[GP1:90,1] + 64.306;
   1:  PR[GP1:91,2] = PR[GP1:90,2] + 23.648;
   1:L PR[91] 10mm/sec CNT100;
   1:  PR[GP1:91,1] = PR[GP1:90,1] + 61.529;
   1:  PR[GP1:91,2] = PR[GP1:90,2] + 25.808;
   1:L PR[91] 10mm/sec CNT100;
   1:  PR[GP1:91,1] = PR[GP1:90,1] + 54.087;
   1:  PR[GP1:91,2] = PR[GP1:90,2] + 31.248;
   1:L PR[91] 10mm/sec CNT100;
   1:  PR[GP1:91,1] = PR[GP1:90,1] + 49.409;
   1:  PR[GP1:91,2] = PR[GP1:90,2] + 32.704;
   1:L PR[91] 10mm/sec CNT100;
   1:  PR[GP1:91,1] = PR[GP1:90,1] + 41.904;
   1:  PR[GP1:91,2] = PR[GP1:90,2] + 34.695;
   1:L PR[91] 10mm/sec CNT100;
   1:  PR[GP1:91,1] = PR[GP1:90,1] + 35.173;
   1:  PR[GP1:91,2] = PR[GP1:90,2] + 34.317;
   1:L PR[91] 10mm/sec CNT100;
   1:  PR[GP1:91,1] = PR[GP1:90,1] + 29.411;
   1:  PR[GP1:91,2] = PR[GP1:90,2] + 33.670;
   1:L PR[91] 10mm/sec CNT100;
   1:  PR[GP1:91,1] = PR[GP1:90,1] + 21.333;
   1:  PR[GP1:91,2] = PR[GP1:90,2] + 30.123;
   1:L PR[91] 10mm/sec CNT100;
   1:  PR[GP1:91,1] = PR[GP1:90,1] + 18.182;
   1:  PR[GP1:91,2] = PR[GP1:90,2] + 28.468;
   1:L PR[91] 10mm/sec CNT100;
   1:  PR[GP1:91,1] = PR[GP1:90,1] + 10.498;
   1:  PR[GP1:91,2] = PR[GP1:90,2] + 20.938;
   1:L PR[91] 10mm/sec CNT100;
   1:  PR[GP1:91,1] = PR[GP1:90,1] + 9.513;
   1:  PR[GP1:91,2] = PR[GP1:90,2] + 19.796;
   1:L PR[91] 10mm/sec CNT100;
   1:  PR[GP1:91,1] = PR[GP1:90,1] + 4.457;
   1:  PR[GP1:91,2] = PR[GP1:90,2] + 8.902;
   1:L PR[91] 10mm/sec CNT100;
   1:  PR[GP1:91,1] = PR[GP1:90,1] + 4.228;
   1:  PR[GP1:91,2] = PR[GP1:90,2] + 8.241;
   1:L PR[91] 10mm/sec CNT100;
   1:  PR[GP1:91,1] = PR[GP1:90,1] + -4.759;
   1:L PR[91] 10mm/sec CNT100;
   1:  PR[GP1:91,1] = PR[GP1:90,1] + -4.990;
   1:  PR[GP1:91,2] = PR[GP1:90,2] + 8.910;
   1:L PR[91] 10mm/sec CNT100;
   1:  PR[GP1:91,1] = PR[GP1:90,1] + -10.049;
   1:  PR[GP1:91,2] = PR[GP1:90,2] + 19.819;
   1:L PR[91] 10mm/sec CNT100;
   1:  PR[GP1:91,1] = PR[GP1:90,1] + -11.035;
   1:  PR[GP1:91,2] = PR[GP1:90,2] + 20.962;
   1:L PR[91] 10mm/sec CNT100;
   1:  PR[GP1:91,1] = PR[GP1:90,1] + -18.719;
   1:  PR[GP1:91,2] = PR[GP1:90,2] + 28.473;
   1:L PR[91] 10mm/sec CNT100;
   1:  PR[GP1:91,1] = PR[GP1:90,1] + -21.872;
   1:  PR[GP1:91,2] = PR[GP1:90,2] + 30.128;
   1:L PR[91] 10mm/sec CNT100;
   1:  PR[GP1:91,1] = PR[GP1:90,1] + -29.947;
   1:  PR[GP1:91,2] = PR[GP1:90,2] + 33.673;
   1:L PR[91] 10mm/sec CNT100;
   1:  PR[GP1:91,1] = PR[GP1:90,1] + -35.710;
   1:  PR[GP1:91,2] = PR[GP1:90,2] + 34.319;
   1:L PR[91] 10mm/sec CNT100;
   1:  PR[GP1:91,1] = PR[GP1:90,1] + -42.437;
   1:  PR[GP1:91,2] = PR[GP1:90,2] + 34.694;
   1:L PR[91] 10mm/sec CNT100;
   1:  PR[GP1:91,1] = PR[GP1:90,1] + -49.942;
   1:  PR[GP1:91,2] = PR[GP1:90,2] + 32.703;
   1:L PR[91] 10mm/sec CNT100;
   1:  PR[GP1:91,1] = PR[GP1:90,1] + -54.617;
   1:  PR[GP1:91,2] = PR[GP1:90,2] + 31.245;
   1:L PR[91] 10mm/sec CNT100;
   1:  PR[GP1:91,1] = PR[GP1:90,1] + -62.059;
   1:  PR[GP1:91,2] = PR[GP1:90,2] + 25.806;
   1:L PR[91] 10mm/sec CNT100;
   1:  PR[GP1:91,1] = PR[GP1:90,1] + -64.835;
   1:  PR[GP1:91,2] = PR[GP1:90,2] + 23.647;
   1:L PR[91] 10mm/sec CNT100;
   1:  PR[GP1:91,1] = PR[GP1:90,1] + -70.247;
   1:  PR[GP1:91,2] = PR[GP1:90,2] + 15.108;
   1:L PR[91] 10mm/sec CNT100;
   1:  PR[GP1:91,1] = PR[GP1:90,1] + -71.633;
   1:  PR[GP1:91,2] = PR[GP1:90,2] + 12.828;
   1:L PR[91] 10mm/sec CNT100;
   1:  PR[GP1:91,1] = PR[GP1:90,1] + -73.659;
   1:  PR[GP1:91,2] = PR[GP1:90,2] + 2.267;
   1:L PR[91] 10mm/sec CNT100;
   1:  PR[GP1:91,1] = PR[GP1:90,1] + -74.025;
   1:  PR[GP1:91,2] = PR[GP1:90,2] + 0.281;
   1:L PR[91] 10mm/sec CNT100;
   1:  PR[GP1:91,1] = PR[GP1:90,1] + -72.062;
   1:  PR[GP1:91,2] = PR[GP1:90,2] + -9.937;
   1:L PR[91] 10mm/sec CNT100;
   1:  PR[GP1:91,1] = PR[GP1:90,1] + -71.632;
   1:  PR[GP1:91,2] = PR[GP1:90,2] + -12.272;
   1:L PR[91] 10mm/sec CNT100;
   1:  PR[GP1:91,1] = PR[GP1:90,1] + -70.247;
   1:  PR[GP1:91,2] = PR[GP1:90,2] + -14.550;
   1:L PR[91] 10mm/sec CNT100;
   1:  PR[GP1:91,1] = PR[GP1:90,1] + -64.835;
   1:  PR[GP1:91,2] = PR[GP1:90,2] + -23.089;
   1:L PR[91] 10mm/sec CNT100;
   1:  PR[GP1:91,1] = PR[GP1:90,1] + -62.059;
   1:  PR[GP1:91,2] = PR[GP1:90,2] + -25.248;
   1:L PR[91] 10mm/sec CNT100;
   1:  PR[GP1:91,1] = PR[GP1:90,1] + -54.617;
   1:  PR[GP1:91,2] = PR[GP1:90,2] + -30.687;
   1:L PR[91] 10mm/sec CNT100;
   1:  PR[GP1:91,1] = PR[GP1:90,1] + -49.942;
   1:  PR[GP1:91,2] = PR[GP1:90,2] + -32.144;
   1:L PR[91] 10mm/sec CNT100;
   1:  PR[GP1:91,1] = PR[GP1:90,1] + -42.437;
   1:  PR[GP1:91,2] = PR[GP1:90,2] + -34.136;
   1:L PR[91] 10mm/sec CNT100;
   1:  PR[GP1:91,1] = PR[GP1:90,1] + -35.709;
   1:  PR[GP1:91,2] = PR[GP1:90,2] + -33.761;
   1:L PR[91] 10mm/sec CNT100;
   1:  PR[GP1:91,1] = PR[GP1:90,1] + -29.947;
   1:  PR[GP1:91,2] = PR[GP1:90,2] + -33.115;
   1:L PR[91] 10mm/sec CNT100;
   1:  PR[GP1:91,1] = PR[GP1:90,1] + -21.872;
   1:  PR[GP1:91,2] = PR[GP1:90,2] + -29.570;
   1:L PR[91] 10mm/sec CNT100;
   1:  PR[GP1:91,1] = PR[GP1:90,1] + -18.719;
   1:  PR[GP1:91,2] = PR[GP1:90,2] + -27.915;
   1:L PR[91] 10mm/sec CNT100;
   1:  PR[GP1:91,1] = PR[GP1:90,1] + -11.035;
   1:  PR[GP1:91,2] = PR[GP1:90,2] + -20.404;
   1:L PR[91] 10mm/sec CNT100;
   1:  PR[GP1:91,1] = PR[GP1:90,1] + -10.049;
   1:  PR[GP1:91,2] = PR[GP1:90,2] + -19.261;
   1:L PR[91] 10mm/sec CNT100;
   1:  PR[GP1:91,1] = PR[GP1:90,1] + -4.988;
   1:  PR[GP1:91,2] = PR[GP1:90,2] + -8.345;
   1:L PR[91] 10mm/sec CNT100;
   1:  PR[GP1:91,1] = PR[GP1:90,1] + -4.759;
   1:  PR[GP1:91,2] = PR[GP1:90,2] + -7.683;
   1:L PR[91] 10mm/sec CNT100;
   1:  PR[GP1:91,1] = PR[GP1:90,1] + 4.228;
   1:L PR[91] 10mm/sec CNT100;
   1:  PR[GP1:91,1] = PR[GP1:90,1] + 7.672;
   1:  PR[GP1:91,2] = PR[GP1:90,2] + -15.458;
   1:  PR[GP1:91,3] = PR[GP1:90,3] + 22.875;
   1:L PR[91] 10mm/sec CNT100;
   1:  PR[GP1:91,1] = PR[GP1:90,1] + 9.538;
   1:  PR[GP1:91,2] = PR[GP1:90,2] + -19.477;
   1:L PR[91] 10mm/sec CNT100;
   1:  PR[GP1:91,1] = PR[GP1:90,1] + 9.778;
   1:  PR[GP1:91,2] = PR[GP1:90,2] + -19.755;
   1:L PR[91] 10mm/sec CNT100;
   1:  PR[GP1:91,1] = PR[GP1:90,1] + 18.246;
   1:  PR[GP1:91,2] = PR[GP1:90,2] + -28.053;
   1:L PR[91] 10mm/sec CNT100;
   1:  PR[GP1:91,1] = PR[GP1:90,1] + 20.446;
   1:  PR[GP1:91,2] = PR[GP1:90,2] + -29.209;
   1:L PR[91] 10mm/sec CNT100;
   1:  PR[GP1:91,1] = PR[GP1:90,1] + 29.472;
   1:  PR[GP1:91,2] = PR[GP1:90,2] + -33.172;
   1:L PR[91] 10mm/sec CNT100;
   1:  PR[GP1:91,1] = PR[GP1:90,1] + 34.254;
   1:  PR[GP1:91,2] = PR[GP1:90,2] + -33.709;
   1:L PR[91] 10mm/sec CNT100;
   1:  PR[GP1:91,1] = PR[GP1:90,1] + 41.938;
   1:  PR[GP1:91,2] = PR[GP1:90,2] + -34.141;
   1:L PR[91] 10mm/sec CNT100;
   1:  PR[GP1:91,1] = PR[GP1:90,1] + 48.578;
   1:  PR[GP1:91,2] = PR[GP1:90,2] + -32.379;
   1:L PR[91] 10mm/sec CNT100;
   1:  PR[GP1:91,1] = PR[GP1:90,1] + 54.085;
   1:  PR[GP1:91,2] = PR[GP1:90,2] + -30.665;
   1:L PR[91] 10mm/sec CNT100;
   1:  PR[GP1:91,1] = PR[GP1:90,1] + 60.872;
   1:  PR[GP1:91,2] = PR[GP1:90,2] + -25.704;
   1:L PR[91] 10mm/sec CNT100;
   1:  PR[GP1:91,1] = PR[GP1:90,1] + 64.271;
   1:  PR[GP1:91,2] = PR[GP1:90,2] + -23.060;
   1:L PR[91] 10mm/sec CNT100;
   1:  PR[GP1:91,1] = PR[GP1:90,1] + 69.285;
   1:  PR[GP1:91,2] = PR[GP1:90,2] + -15.153;
   1:L PR[91] 10mm/sec CNT100;
   1:  PR[GP1:91,1] = PR[GP1:90,1] + 71.048;
   1:  PR[GP1:91,2] = PR[GP1:90,2] + -12.256;
   1:L PR[91] 10mm/sec CNT100;
   1:  PR[GP1:91,1] = PR[GP1:90,1] + 72.939;
   1:  PR[GP1:91,2] = PR[GP1:90,2] + -2.397;
   1:L PR[91] 10mm/sec CNT100;
   1:  PR[GP1:91,1] = PR[GP1:90,1] + 73.433;
   1:  PR[GP1:91,2] = PR[GP1:90,2] + 0.277;
   1:L PR[91] 10mm/sec CNT100;
   1:  PR[GP1:91,1] = PR[GP1:90,1] + 71.595;
   1:  PR[GP1:91,2] = PR[GP1:90,2] + 9.842;
   1:L PR[91] 10mm/sec CNT100;
   1:  PR[GP1:91,1] = PR[GP1:90,1] + 71.047;
   1:  PR[GP1:91,2] = PR[GP1:90,2] + 12.816;
   1:L PR[91] 10mm/sec CNT100;
   1:  PR[GP1:91,1] = PR[GP1:90,1] + 69.285;
   1:  PR[GP1:91,2] = PR[GP1:90,2] + 15.711;
   1:L PR[91] 10mm/sec CNT100;
   1:  PR[GP1:91,1] = PR[GP1:90,1] + 64.271;
   1:  PR[GP1:91,2] = PR[GP1:90,2] + 23.618;
   1:L PR[91] 10mm/sec CNT100;
   1:  PR[GP1:91,1] = PR[GP1:90,1] + 60.872;
   1:  PR[GP1:91,2] = PR[GP1:90,2] + 26.262;
   1:L PR[91] 10mm/sec CNT100;
   1:  PR[GP1:91,1] = PR[GP1:90,1] + 54.085;
   1:  PR[GP1:91,2] = PR[GP1:90,2] + 31.223;
   1:L PR[91] 10mm/sec CNT100;
   1:  PR[GP1:91,1] = PR[GP1:90,1] + 48.578;
   1:  PR[GP1:91,2] = PR[GP1:90,2] + 32.937;
   1:L PR[91] 10mm/sec CNT100;
   1:  PR[GP1:91,1] = PR[GP1:90,1] + 41.938;
   1:  PR[GP1:91,2] = PR[GP1:90,2] + 34.699;
   1:L PR[91] 10mm/sec CNT100;
   1:  PR[GP1:91,1] = PR[GP1:90,1] + 34.254;
   1:  PR[GP1:91,2] = PR[GP1:90,2] + 34.267;
   1:L PR[91] 10mm/sec CNT100;
   1:  PR[GP1:91,1] = PR[GP1:90,1] + 29.472;
   1:  PR[GP1:91,2] = PR[GP1:90,2] + 33.730;
   1:L PR[91] 10mm/sec CNT100;
   1:  PR[GP1:91,1] = PR[GP1:90,1] + 20.446;
   1:  PR[GP1:91,2] = PR[GP1:90,2] + 29.767;
   1:L PR[91] 10mm/sec CNT100;
   1:  PR[GP1:91,1] = PR[GP1:90,1] + 18.246;
   1:  PR[GP1:91,2] = PR[GP1:90,2] + 28.611;
   1:L PR[91] 10mm/sec CNT100;
   1:  PR[GP1:91,1] = PR[GP1:90,1] + 9.778;
   1:  PR[GP1:91,2] = PR[GP1:90,2] + 20.313;
   1:L PR[91] 10mm/sec CNT100;
   1:  PR[GP1:91,1] = PR[GP1:90,1] + 9.538;
   1:  PR[GP1:91,2] = PR[GP1:90,2] + 20.035;
   1:L PR[91] 10mm/sec CNT100;
   1:  PR[GP1:91,1] = PR[GP1:90,1] + 7.683;
   1:  PR[GP1:91,2] = PR[GP1:90,2] + 16.040;
   1:L PR[91] 10mm/sec CNT100;
   1:  PR[GP1:91,1] = PR[GP1:90,1] + 4.092;
   1:  PR[GP1:91,2] = PR[GP1:90,2] + 8.566;
   1:L PR[91] 10mm/sec CNT100;
   1:  PR[GP1:91,1] = PR[GP1:90,1] + -4.630;
   1:L PR[91] 10mm/sec CNT100;
   1:  PR[GP1:91,1] = PR[GP1:90,1] + -8.200;
   1:  PR[GP1:91,2] = PR[GP1:90,2] + 16.018;
   1:L PR[91] 10mm/sec CNT100;
   1:  PR[GP1:91,1] = PR[GP1:90,1] + -10.074;
   1:  PR[GP1:91,2] = PR[GP1:90,2] + 20.059;
   1:L PR[91] 10mm/sec CNT100;
   1:  PR[GP1:91,1] = PR[GP1:90,1] + -10.315;
   1:  PR[GP1:91,2] = PR[GP1:90,2] + 20.339;
   1:L PR[91] 10mm/sec CNT100;
   1:  PR[GP1:91,1] = PR[GP1:90,1] + -18.783;
   1:  PR[GP1:91,2] = PR[GP1:90,2] + 28.616;
   1:L PR[91] 10mm/sec CNT100;
   1:  PR[GP1:91,1] = PR[GP1:90,1] + -20.986;
   1:  PR[GP1:91,2] = PR[GP1:90,2] + 29.772;
   1:L PR[91] 10mm/sec CNT100;
   1:  PR[GP1:91,1] = PR[GP1:90,1] + -30.009;
   1:  PR[GP1:91,2] = PR[GP1:90,2] + 33.733;
   1:L PR[91] 10mm/sec CNT100;
   1:  PR[GP1:91,1] = PR[GP1:90,1] + -34.792;
   1:  PR[GP1:91,2] = PR[GP1:90,2] + 34.269;
   1:L PR[91] 10mm/sec CNT100;
   1:  PR[GP1:91,1] = PR[GP1:90,1] + -42.471;
   1:  PR[GP1:91,2] = PR[GP1:90,2] + 34.698;
   1:L PR[91] 10mm/sec CNT100;
   1:  PR[GP1:91,1] = PR[GP1:90,1] + -49.112;
   1:  PR[GP1:91,2] = PR[GP1:90,2] + 32.935;
   1:L PR[91] 10mm/sec CNT100;
   1:  PR[GP1:91,1] = PR[GP1:90,1] + -54.615;
   1:  PR[GP1:91,2] = PR[GP1:90,2] + 31.220;
   1:L PR[91] 10mm/sec CNT100;
   1:  PR[GP1:91,1] = PR[GP1:90,1] + -61.401;
   1:  PR[GP1:91,2] = PR[GP1:90,2] + 26.260;
   1:L PR[91] 10mm/sec CNT100;
   1:  PR[GP1:91,1] = PR[GP1:90,1] + -64.799;
   1:  PR[GP1:91,2] = PR[GP1:90,2] + 23.617;
   1:L PR[91] 10mm/sec CNT100;
   1:  PR[GP1:91,1] = PR[GP1:90,1] + -69.812;
   1:  PR[GP1:91,2] = PR[GP1:90,2] + 15.708;
   1:L PR[91] 10mm/sec CNT100;
   1:  PR[GP1:91,1] = PR[GP1:90,1] + -71.575;
   1:  PR[GP1:91,2] = PR[GP1:90,2] + 12.808;
   1:L PR[91] 10mm/sec CNT100;
   1:  PR[GP1:91,1] = PR[GP1:90,1] + -73.466;
   1:  PR[GP1:91,2] = PR[GP1:90,2] + 2.952;
   1:L PR[91] 10mm/sec CNT100;
   1:  PR[GP1:91,1] = PR[GP1:90,1] + -73.959;
   1:  PR[GP1:91,2] = PR[GP1:90,2] + 0.281;
   1:L PR[91] 10mm/sec CNT100;
   1:  PR[GP1:91,1] = PR[GP1:90,1] + -72.122;
   1:  PR[GP1:91,2] = PR[GP1:90,2] + -9.281;
   1:L PR[91] 10mm/sec CNT100;
   1:  PR[GP1:91,1] = PR[GP1:90,1] + -71.574;
   1:  PR[GP1:91,2] = PR[GP1:90,2] + -12.252;
   1:L PR[91] 10mm/sec CNT100;
   1:  PR[GP1:91,1] = PR[GP1:90,1] + -69.812;
   1:  PR[GP1:91,2] = PR[GP1:90,2] + -15.150;
   1:L PR[91] 10mm/sec CNT100;
   1:  PR[GP1:91,1] = PR[GP1:90,1] + -64.799;
   1:  PR[GP1:91,2] = PR[GP1:90,2] + -23.059;
   1:L PR[91] 10mm/sec CNT100;
   1:  PR[GP1:91,1] = PR[GP1:90,1] + -61.401;
   1:  PR[GP1:91,2] = PR[GP1:90,2] + -25.702;
   1:L PR[91] 10mm/sec CNT100;
   1:  PR[GP1:91,1] = PR[GP1:90,1] + -54.615;
   1:  PR[GP1:91,2] = PR[GP1:90,2] + -30.662;
   1:L PR[91] 10mm/sec CNT100;
   1:  PR[GP1:91,1] = PR[GP1:90,1] + -49.112;
   1:  PR[GP1:91,2] = PR[GP1:90,2] + -32.377;
   1:L PR[91] 10mm/sec CNT100;
   1:  PR[GP1:91,1] = PR[GP1:90,1] + -42.471;
   1:  PR[GP1:91,2] = PR[GP1:90,2] + -34.139;
   1:L PR[91] 10mm/sec CNT100;
   1:  PR[GP1:91,1] = PR[GP1:90,1] + -34.792;
   1:  PR[GP1:91,2] = PR[GP1:90,2] + -33.711;
   1:L PR[91] 10mm/sec CNT100;
   1:  PR[GP1:91,1] = PR[GP1:90,1] + -30.008;
   1:  PR[GP1:91,2] = PR[GP1:90,2] + -33.175;
   1:L PR[91] 10mm/sec CNT100;
   1:  PR[GP1:91,1] = PR[GP1:90,1] + -20.986;
   1:  PR[GP1:91,2] = PR[GP1:90,2] + -29.214;
   1:L PR[91] 10mm/sec CNT100;
   1:  PR[GP1:91,1] = PR[GP1:90,1] + -18.783;
   1:  PR[GP1:91,2] = PR[GP1:90,2] + -28.058;
   1:L PR[91] 10mm/sec CNT100;
   1:  PR[GP1:91,1] = PR[GP1:90,1] + -10.315;
   1:  PR[GP1:91,2] = PR[GP1:90,2] + -19.781;
   1:L PR[91] 10mm/sec CNT100;
   1:  PR[GP1:91,1] = PR[GP1:90,1] + -10.074;
   1:  PR[GP1:91,2] = PR[GP1:90,2] + -19.501;
   1:L PR[91] 10mm/sec CNT100;
   1:  PR[GP1:91,1] = PR[GP1:90,1] + -8.211;
   1:  PR[GP1:91,2] = PR[GP1:90,2] + -15.484;
   1:L PR[91] 10mm/sec CNT100;
   1:  PR[GP1:91,1] = PR[GP1:90,1] + -4.623;
   1:  PR[GP1:91,2] = PR[GP1:90,2] + -8.008;
   1:L PR[91] 10mm/sec CNT100;
   1:  PR[GP1:91,1] = PR[GP1:90,1] + 4.098;
   1:L PR[91] 10mm/sec CNT100;
   1:  PR[GP1:91,1] = PR[GP1:90,1] + 9.214;
   1:  PR[GP1:91,2] = PR[GP1:90,2] + -19.187;
   1:  PR[GP1:91,3] = PR[GP1:90,3] + 23.485;
   1:L PR[91] 10mm/sec CNT100;
   1:  PR[GP1:91,1] = PR[GP1:90,1] + 9.502;
   1:  PR[GP1:91,2] = PR[GP1:90,2] + -19.662;
   1:L PR[91] 10mm/sec CNT100;
   1:  PR[GP1:91,1] = PR[GP1:90,1] + 12.076;
   1:  PR[GP1:91,2] = PR[GP1:90,2] + -22.088;
   1:L PR[91] 10mm/sec CNT100;
   1:  PR[GP1:91,1] = PR[GP1:90,1] + 18.309;
   1:  PR[GP1:91,2] = PR[GP1:90,2] + -28.196;
   1:L PR[91] 10mm/sec CNT100;
   1:  PR[GP1:91,1] = PR[GP1:90,1] + 19.559;
   1:  PR[GP1:91,2] = PR[GP1:90,2] + -28.852;
   1:L PR[91] 10mm/sec CNT100;
   1:  PR[GP1:91,1] = PR[GP1:90,1] + 29.533;
   1:  PR[GP1:91,2] = PR[GP1:90,2] + -33.232;
   1:L PR[91] 10mm/sec CNT100;
   1:  PR[GP1:91,1] = PR[GP1:90,1] + 33.336;
   1:  PR[GP1:91,2] = PR[GP1:90,2] + -33.659;
   1:L PR[91] 10mm/sec CNT100;
   1:  PR[GP1:91,1] = PR[GP1:90,1] + 41.972;
   1:  PR[GP1:91,2] = PR[GP1:90,2] + -34.144;
   1:L PR[91] 10mm/sec CNT100;
   1:  PR[GP1:91,1] = PR[GP1:90,1] + 47.748;
   1:  PR[GP1:91,2] = PR[GP1:90,2] + -32.612;
   1:L PR[91] 10mm/sec CNT100;
   1:  PR[GP1:91,1] = PR[GP1:90,1] + 54.083;
   1:  PR[GP1:91,2] = PR[GP1:90,2] + -30.639;
   1:L PR[91] 10mm/sec CNT100;
   1:  PR[GP1:91,1] = PR[GP1:90,1] + 60.214;
   1:  PR[GP1:91,2] = PR[GP1:90,2] + -26.158;
   1:L PR[91] 10mm/sec CNT100;
   1:  PR[GP1:91,1] = PR[GP1:90,1] + 64.236;
   1:  PR[GP1:91,2] = PR[GP1:90,2] + -23.029;
   1:L PR[91] 10mm/sec CNT100;
   1:  PR[GP1:91,1] = PR[GP1:90,1] + 68.850;
   1:  PR[GP1:91,2] = PR[GP1:90,2] + -15.752;
   1:L PR[91] 10mm/sec CNT100;
   1:  PR[GP1:91,1] = PR[GP1:90,1] + 70.990;
   1:  PR[GP1:91,2] = PR[GP1:90,2] + -12.237;
   1:L PR[91] 10mm/sec CNT100;
   1:  PR[GP1:91,1] = PR[GP1:90,1] + 72.746;
   1:  PR[GP1:91,2] = PR[GP1:90,2] + -3.082;
   1:L PR[91] 10mm/sec CNT100;
   1:  PR[GP1:91,1] = PR[GP1:90,1] + 73.366;
   1:  PR[GP1:91,2] = PR[GP1:90,2] + 0.277;
   1:L PR[91] 10mm/sec CNT100;
   1:  PR[GP1:91,1] = PR[GP1:90,1] + 71.655;
   1:  PR[GP1:91,2] = PR[GP1:90,2] + 9.186;
   1:L PR[91] 10mm/sec CNT100;
   1:  PR[GP1:91,1] = PR[GP1:90,1] + 70.989;
   1:  PR[GP1:91,2] = PR[GP1:90,2] + 12.797;
   1:L PR[91] 10mm/sec CNT100;
   1:  PR[GP1:91,1] = PR[GP1:90,1] + 68.850;
   1:  PR[GP1:91,2] = PR[GP1:90,2] + 16.310;
   1:L PR[91] 10mm/sec CNT100;
   1:  PR[GP1:91,1] = PR[GP1:90,1] + 64.236;
   1:  PR[GP1:91,2] = PR[GP1:90,2] + 23.587;
   1:L PR[91] 10mm/sec CNT100;
   1:  PR[GP1:91,1] = PR[GP1:90,1] + 60.214;
   1:  PR[GP1:91,2] = PR[GP1:90,2] + 26.716;
   1:L PR[91] 10mm/sec CNT100;
   1:  PR[GP1:91,1] = PR[GP1:90,1] + 54.082;
   1:  PR[GP1:91,2] = PR[GP1:90,2] + 31.198;
   1:L PR[91] 10mm/sec CNT100;
   1:  PR[GP1:91,1] = PR[GP1:90,1] + 47.748;
   1:  PR[GP1:91,2] = PR[GP1:90,2] + 33.170;
   1:L PR[91] 10mm/sec CNT100;
   1:  PR[GP1:91,1] = PR[GP1:90,1] + 41.972;
   1:  PR[GP1:91,2] = PR[GP1:90,2] + 34.702;
   1:L PR[91] 10mm/sec CNT100;
   1:  PR[GP1:91,1] = PR[GP1:90,1] + 33.336;
   1:  PR[GP1:91,2] = PR[GP1:90,2] + 34.217;
   1:L PR[91] 10mm/sec CNT100;
   1:  PR[GP1:91,1] = PR[GP1:90,1] + 29.533;
   1:  PR[GP1:91,2] = PR[GP1:90,2] + 33.790;
   1:L PR[91] 10mm/sec CNT100;
   1:  PR[GP1:91,1] = PR[GP1:90,1] + 19.559;
   1:  PR[GP1:91,2] = PR[GP1:90,2] + 29.410;
   1:L PR[91] 10mm/sec CNT100;
   1:  PR[GP1:91,1] = PR[GP1:90,1] + 18.309;
   1:  PR[GP1:91,2] = PR[GP1:90,2] + 28.754;
   1:L PR[91] 10mm/sec CNT100;
   1:  PR[GP1:91,1] = PR[GP1:90,1] + 12.076;
   1:  PR[GP1:91,2] = PR[GP1:90,2] + 22.646;
   1:L PR[91] 10mm/sec CNT100;
   1:  PR[GP1:91,1] = PR[GP1:90,1] + 9.502;
   1:  PR[GP1:91,2] = PR[GP1:90,2] + 20.220;
   1:L PR[91] 10mm/sec CNT100;
   1:  PR[GP1:91,1] = PR[GP1:90,1] + 9.214;
   1:  PR[GP1:91,2] = PR[GP1:90,2] + 19.745;
   1:L PR[91] 10mm/sec CNT100;
   1:  PR[GP1:91,1] = PR[GP1:90,1] + 3.998;
   1:  PR[GP1:91,2] = PR[GP1:90,2] + 8.891;
   1:L PR[91] 10mm/sec CNT100;
   1:  PR[GP1:91,1] = PR[GP1:90,1] + -4.546;
   1:L PR[91] 10mm/sec CNT100;
   1:  PR[GP1:91,1] = PR[GP1:90,1] + -9.752;
   1:  PR[GP1:91,2] = PR[GP1:90,2] + 19.771;
   1:L PR[91] 10mm/sec CNT100;
   1:  PR[GP1:91,1] = PR[GP1:90,1] + -10.039;
   1:  PR[GP1:91,2] = PR[GP1:90,2] + 20.245;
   1:L PR[91] 10mm/sec CNT100;
   1:  PR[GP1:91,1] = PR[GP1:90,1] + -12.602;
   1:  PR[GP1:91,2] = PR[GP1:90,2] + 22.654;
   1:L PR[91] 10mm/sec CNT100;
   1:  PR[GP1:91,1] = PR[GP1:90,1] + -18.847;
   1:  PR[GP1:91,2] = PR[GP1:90,2] + 28.759;
   1:L PR[91] 10mm/sec CNT100;
   1:  PR[GP1:91,1] = PR[GP1:90,1] + -20.100;
   1:  PR[GP1:91,2] = PR[GP1:90,2] + 29.416;
   1:L PR[91] 10mm/sec CNT100;
   1:  PR[GP1:91,1] = PR[GP1:90,1] + -30.070;
   1:  PR[GP1:91,2] = PR[GP1:90,2] + 33.794;
   1:L PR[91] 10mm/sec CNT100;
   1:  PR[GP1:91,1] = PR[GP1:90,1] + -33.874;
   1:  PR[GP1:91,2] = PR[GP1:90,2] + 34.220;
   1:L PR[91] 10mm/sec CNT100;
   1:  PR[GP1:91,1] = PR[GP1:90,1] + -42.506;
   1:  PR[GP1:91,2] = PR[GP1:90,2] + 34.701;
   1:L PR[91] 10mm/sec CNT100;
   1:  PR[GP1:91,1] = PR[GP1:90,1] + -48.282;
   1:  PR[GP1:91,2] = PR[GP1:90,2] + 33.168;
   1:L PR[91] 10mm/sec CNT100;
   1:  PR[GP1:91,1] = PR[GP1:90,1] + -54.613;
   1:  PR[GP1:91,2] = PR[GP1:90,2] + 31.195;
   1:L PR[91] 10mm/sec CNT100;
   1:  PR[GP1:91,1] = PR[GP1:90,1] + -60.744;
   1:  PR[GP1:91,2] = PR[GP1:90,2] + 26.714;
   1:L PR[91] 10mm/sec CNT100;
   1:  PR[GP1:91,1] = PR[GP1:90,1] + -64.764;
   1:  PR[GP1:91,2] = PR[GP1:90,2] + 23.587;
   1:L PR[91] 10mm/sec CNT100;
   1:  PR[GP1:91,1] = PR[GP1:90,1] + -69.378;
   1:  PR[GP1:91,2] = PR[GP1:90,2] + 16.308;
   1:L PR[91] 10mm/sec CNT100;
   1:  PR[GP1:91,1] = PR[GP1:90,1] + -71.517;
   1:  PR[GP1:91,2] = PR[GP1:90,2] + 12.789;
   1:L PR[91] 10mm/sec CNT100;
   1:  PR[GP1:91,1] = PR[GP1:90,1] + -73.273;
   1:  PR[GP1:91,2] = PR[GP1:90,2] + 3.636;
   1:L PR[91] 10mm/sec CNT100;
   1:  PR[GP1:91,1] = PR[GP1:90,1] + -73.892;
   1:  PR[GP1:91,2] = PR[GP1:90,2] + 0.281;
   1:L PR[91] 10mm/sec CNT100;
   1:  PR[GP1:91,1] = PR[GP1:90,1] + -72.181;
   1:  PR[GP1:91,2] = PR[GP1:90,2] + -8.625;
   1:L PR[91] 10mm/sec CNT100;
   1:  PR[GP1:91,1] = PR[GP1:90,1] + -71.516;
   1:  PR[GP1:91,2] = PR[GP1:90,2] + -12.232;
   1:L PR[91] 10mm/sec CNT100;
   1:  PR[GP1:91,1] = PR[GP1:90,1] + -69.378;
   1:  PR[GP1:91,2] = PR[GP1:90,2] + -15.749;
   1:L PR[91] 10mm/sec CNT100;
   1:  PR[GP1:91,1] = PR[GP1:90,1] + -64.764;
   1:  PR[GP1:91,2] = PR[GP1:90,2] + -23.029;
   1:L PR[91] 10mm/sec CNT100;
   1:  PR[GP1:91,1] = PR[GP1:90,1] + -60.744;
   1:  PR[GP1:91,2] = PR[GP1:90,2] + -26.156;
   1:L PR[91] 10mm/sec CNT100;
   1:  PR[GP1:91,1] = PR[GP1:90,1] + -54.613;
   1:  PR[GP1:91,2] = PR[GP1:90,2] + -30.637;
   1:L PR[91] 10mm/sec CNT100;
   1:  PR[GP1:91,1] = PR[GP1:90,1] + -48.282;
   1:  PR[GP1:91,2] = PR[GP1:90,2] + -32.610;
   1:L PR[91] 10mm/sec CNT100;
   1:  PR[GP1:91,1] = PR[GP1:90,1] + -42.505;
   1:  PR[GP1:91,2] = PR[GP1:90,2] + -34.143;
   1:L PR[91] 10mm/sec CNT100;
   1:  PR[GP1:91,1] = PR[GP1:90,1] + -33.874;
   1:  PR[GP1:91,2] = PR[GP1:90,2] + -33.662;
   1:L PR[91] 10mm/sec CNT100;
   1:  PR[GP1:91,1] = PR[GP1:90,1] + -30.070;
   1:  PR[GP1:91,2] = PR[GP1:90,2] + -33.236;
   1:L PR[91] 10mm/sec CNT100;
   1:  PR[GP1:91,1] = PR[GP1:90,1] + -20.099;
   1:  PR[GP1:91,2] = PR[GP1:90,2] + -28.858;
   1:L PR[91] 10mm/sec CNT100;
   1:  PR[GP1:91,1] = PR[GP1:90,1] + -18.847;
   1:  PR[GP1:91,2] = PR[GP1:90,2] + -28.201;
   1:L PR[91] 10mm/sec CNT100;
   1:  PR[GP1:91,1] = PR[GP1:90,1] + -12.602;
   1:  PR[GP1:91,2] = PR[GP1:90,2] + -22.096;
   1:L PR[91] 10mm/sec CNT100;
   1:  PR[GP1:91,1] = PR[GP1:90,1] + -10.039;
   1:  PR[GP1:91,2] = PR[GP1:90,2] + -19.686;
   1:L PR[91] 10mm/sec CNT100;
   1:  PR[GP1:91,1] = PR[GP1:90,1] + -9.752;
   1:  PR[GP1:91,2] = PR[GP1:90,2] + -19.213;
   1:L PR[91] 10mm/sec CNT100;
   1:  PR[GP1:91,1] = PR[GP1:90,1] + -4.530;
   1:  PR[GP1:91,2] = PR[GP1:90,2] + -8.333;
   1:L PR[91] 10mm/sec CNT100;
   1:  PR[GP1:91,1] = PR[GP1:90,1] + 4.014;
   1:L PR[91] 10mm/sec CNT100;
   1:  PR[GP1:91,1] = PR[GP1:90,1] + 8.608;
   1:  PR[GP1:91,2] = PR[GP1:90,2] + -18.445;
   1:  PR[GP1:91,3] = PR[GP1:90,3] + 24.095;
   1:L PR[91] 10mm/sec CNT100;
   1:  PR[GP1:91,1] = PR[GP1:90,1] + 9.490;
   1:  PR[GP1:91,2] = PR[GP1:90,2] + -19.900;
   1:L PR[91] 10mm/sec CNT100;
   1:  PR[GP1:91,1] = PR[GP1:90,1] + 16.581;
   1:  PR[GP1:91,2] = PR[GP1:90,2] + -26.583;
   1:L PR[91] 10mm/sec CNT100;
   1:  PR[GP1:91,1] = PR[GP1:90,1] + 18.373;
   1:  PR[GP1:91,2] = PR[GP1:90,2] + -28.339;
   1:L PR[91] 10mm/sec CNT100;
   1:  PR[GP1:91,1] = PR[GP1:90,1] + 18.672;
   1:  PR[GP1:91,2] = PR[GP1:90,2] + -28.496;
   1:L PR[91] 10mm/sec CNT100;
   1:  PR[GP1:91,1] = PR[GP1:90,1] + 29.595;
   1:  PR[GP1:91,2] = PR[GP1:90,2] + -33.292;
   1:L PR[91] 10mm/sec CNT100;
   1:  PR[GP1:91,1] = PR[GP1:90,1] + 32.417;
   1:  PR[GP1:91,2] = PR[GP1:90,2] + -33.609;
   1:L PR[91] 10mm/sec CNT100;
   1:  PR[GP1:91,1] = PR[GP1:90,1] + 42.006;
   1:  PR[GP1:91,2] = PR[GP1:90,2] + -34.148;
   1:L PR[91] 10mm/sec CNT100;
   1:  PR[GP1:91,1] = PR[GP1:90,1] + 46.917;
   1:  PR[GP1:91,2] = PR[GP1:90,2] + -32.845;
   1:L PR[91] 10mm/sec CNT100;
   1:  PR[GP1:91,1] = PR[GP1:90,1] + 54.080;
   1:  PR[GP1:91,2] = PR[GP1:90,2] + -30.614;
   1:L PR[91] 10mm/sec CNT100;
   1:  PR[GP1:91,1] = PR[GP1:90,1] + 59.557;
   1:  PR[GP1:91,2] = PR[GP1:90,2] + -26.612;
   1:L PR[91] 10mm/sec CNT100;
   1:  PR[GP1:91,1] = PR[GP1:90,1] + 64.201;
   1:  PR[GP1:91,2] = PR[GP1:90,2] + -22.999;
   1:L PR[91] 10mm/sec CNT100;
   1:  PR[GP1:91,1] = PR[GP1:90,1] + 68.415;
   1:  PR[GP1:91,2] = PR[GP1:90,2] + -16.352;
   1:L PR[91] 10mm/sec CNT100;
   1:  PR[GP1:91,1] = PR[GP1:90,1] + 70.932;
   1:  PR[GP1:91,2] = PR[GP1:90,2] + -12.218;
   1:L PR[91] 10mm/sec CNT100;
   1:  PR[GP1:91,1] = PR[GP1:90,1] + 72.553;
   1:  PR[GP1:91,2] = PR[GP1:90,2] + -3.767;
   1:L PR[91] 10mm/sec CNT100;
   1:  PR[GP1:91,1] = PR[GP1:90,1] + 73.300;
   1:  PR[GP1:91,2] = PR[GP1:90,2] + 0.277;
   1:L PR[91] 10mm/sec CNT100;
   1:  PR[GP1:91,1] = PR[GP1:90,1] + 71.714;
   1:  PR[GP1:91,2] = PR[GP1:90,2] + 8.529;
   1:L PR[91] 10mm/sec CNT100;
   1:  PR[GP1:91,1] = PR[GP1:90,1] + 70.931;
   1:  PR[GP1:91,2] = PR[GP1:90,2] + 12.778;
   1:L PR[91] 10mm/sec CNT100;
   1:  PR[GP1:91,1] = PR[GP1:90,1] + 68.415;
   1:  PR[GP1:91,2] = PR[GP1:90,2] + 16.910;
   1:L PR[91] 10mm/sec CNT100;
   1:  PR[GP1:91,1] = PR[GP1:90,1] + 64.200;
   1:  PR[GP1:91,2] = PR[GP1:90,2] + 23.557;
   1:L PR[91] 10mm/sec CNT100;
   1:  PR[GP1:91,1] = PR[GP1:90,1] + 59.557;
   1:  PR[GP1:91,2] = PR[GP1:90,2] + 27.170;
   1:L PR[91] 10mm/sec CNT100;
   1:  PR[GP1:91,1] = PR[GP1:90,1] + 54.080;
   1:  PR[GP1:91,2] = PR[GP1:90,2] + 31.172;
   1:L PR[91] 10mm/sec CNT100;
   1:  PR[GP1:91,1] = PR[GP1:90,1] + 46.917;
   1:  PR[GP1:91,2] = PR[GP1:90,2] + 33.403;
   1:L PR[91] 10mm/sec CNT100;
   1:  PR[GP1:91,1] = PR[GP1:90,1] + 42.006;
   1:  PR[GP1:91,2] = PR[GP1:90,2] + 34.706;
   1:L PR[91] 10mm/sec CNT100;
   1:  PR[GP1:91,1] = PR[GP1:90,1] + 32.417;
   1:  PR[GP1:91,2] = PR[GP1:90,2] + 34.167;
   1:L PR[91] 10mm/sec CNT100;
   1:  PR[GP1:91,1] = PR[GP1:90,1] + 29.594;
   1:  PR[GP1:91,2] = PR[GP1:90,2] + 33.850;
   1:L PR[91] 10mm/sec CNT100;
   1:  PR[GP1:91,1] = PR[GP1:90,1] + 18.672;
   1:  PR[GP1:91,2] = PR[GP1:90,2] + 29.054;
   1:L PR[91] 10mm/sec CNT100;
   1:  PR[GP1:91,1] = PR[GP1:90,1] + 18.373;
   1:  PR[GP1:91,2] = PR[GP1:90,2] + 28.897;
   1:L PR[91] 10mm/sec CNT100;
   1:  PR[GP1:91,1] = PR[GP1:90,1] + 16.581;
   1:  PR[GP1:91,2] = PR[GP1:90,2] + 27.141;
   1:L PR[91] 10mm/sec CNT100;
   1:  PR[GP1:91,1] = PR[GP1:90,1] + 9.490;
   1:  PR[GP1:91,2] = PR[GP1:90,2] + 20.458;
   1:L PR[91] 10mm/sec CNT100;
   1:  PR[GP1:91,1] = PR[GP1:90,1] + 8.607;
   1:  PR[GP1:91,2] = PR[GP1:90,2] + 19.002;
   1:L PR[91] 10mm/sec CNT100;
   1:  PR[GP1:91,1] = PR[GP1:90,1] + 3.904;
   1:  PR[GP1:91,2] = PR[GP1:90,2] + 9.216;
   1:L PR[91] 10mm/sec CNT100;
   1:  PR[GP1:91,1] = PR[GP1:90,1] + -4.454;
   1:L PR[91] 10mm/sec CNT100;
   1:  PR[GP1:91,1] = PR[GP1:90,1] + -9.145;
   1:  PR[GP1:91,2] = PR[GP1:90,2] + 19.026;
   1:L PR[91] 10mm/sec CNT100;
   1:  PR[GP1:91,1] = PR[GP1:90,1] + -10.026;
   1:  PR[GP1:91,2] = PR[GP1:90,2] + 20.481;
   1:L PR[91] 10mm/sec CNT100;
   1:  PR[GP1:91,1] = PR[GP1:90,1] + -17.107;
   1:  PR[GP1:91,2] = PR[GP1:90,2] + 27.139;
   1:L PR[91] 10mm/sec CNT100;
   1:  PR[GP1:91,1] = PR[GP1:90,1] + -18.911;
   1:  PR[GP1:91,2] = PR[GP1:90,2] + 28.902;
   1:L PR[91] 10mm/sec CNT100;
   1:  PR[GP1:91,1] = PR[GP1:90,1] + -19.213;
   1:  PR[GP1:91,2] = PR[GP1:90,2] + 29.061;
   1:L PR[91] 10mm/sec CNT100;
   1:  PR[GP1:91,1] = PR[GP1:90,1] + -30.132;
   1:  PR[GP1:91,2] = PR[GP1:90,2] + 33.854;
   1:L PR[91] 10mm/sec CNT100;
   1:  PR[GP1:91,1] = PR[GP1:90,1] + -32.956;
   1:  PR[GP1:91,2] = PR[GP1:90,2] + 34.170;
   1:L PR[91] 10mm/sec CNT100;
   1:  PR[GP1:91,1] = PR[GP1:90,1] + -42.540;
   1:  PR[GP1:91,2] = PR[GP1:90,2] + 34.704;
   1:L PR[91] 10mm/sec CNT100;
   1:  PR[GP1:91,1] = PR[GP1:90,1] + -47.452;
   1:  PR[GP1:91,2] = PR[GP1:90,2] + 33.401;
   1:L PR[91] 10mm/sec CNT100;
   1:  PR[GP1:91,1] = PR[GP1:90,1] + -54.611;
   1:  PR[GP1:91,2] = PR[GP1:90,2] + 31.170;
   1:L PR[91] 10mm/sec CNT100;
   1:  PR[GP1:91,1] = PR[GP1:90,1] + -60.087;
   1:  PR[GP1:91,2] = PR[GP1:90,2] + 27.167;
   1:L PR[91] 10mm/sec CNT100;
   1:  PR[GP1:91,1] = PR[GP1:90,1] + -64.729;
   1:  PR[GP1:91,2] = PR[GP1:90,2] + 23.556;
   1:L PR[91] 10mm/sec CNT100;
   1:  PR[GP1:91,1] = PR[GP1:90,1] + -68.943;
   1:  PR[GP1:91,2] = PR[GP1:90,2] + 16.907;
   1:L PR[91] 10mm/sec CNT100;
   1:  PR[GP1:91,1] = PR[GP1:90,1] + -71.459;
   1:  PR[GP1:91,2] = PR[GP1:90,2] + 12.769;
   1:L PR[91] 10mm/sec CNT100;
   1:  PR[GP1:91,1] = PR[GP1:90,1] + -73.080;
   1:  PR[GP1:91,2] = PR[GP1:90,2] + 4.320;
   1:L PR[91] 10mm/sec CNT100;
   1:  PR[GP1:91,1] = PR[GP1:90,1] + -73.826;
   1:  PR[GP1:91,2] = PR[GP1:90,2] + 0.281;
   1:L PR[91] 10mm/sec CNT100;
   1:  PR[GP1:91,1] = PR[GP1:90,1] + -72.241;
   1:  PR[GP1:91,2] = PR[GP1:90,2] + -7.969;
   1:L PR[91] 10mm/sec CNT100;
   1:  PR[GP1:91,1] = PR[GP1:90,1] + -71.458;
   1:  PR[GP1:91,2] = PR[GP1:90,2] + -12.213;
   1:L PR[91] 10mm/sec CNT100;
   1:  PR[GP1:91,1] = PR[GP1:90,1] + -68.943;
   1:  PR[GP1:91,2] = PR[GP1:90,2] + -16.349;
   1:L PR[91] 10mm/sec CNT100;
   1:  PR[GP1:91,1] = PR[GP1:90,1] + -64.729;
   1:  PR[GP1:91,2] = PR[GP1:90,2] + -22.998;
   1:L PR[91] 10mm/sec CNT100;
   1:  PR[GP1:91,1] = PR[GP1:90,1] + -60.087;
   1:  PR[GP1:91,2] = PR[GP1:90,2] + -26.609;
   1:L PR[91] 10mm/sec CNT100;
   1:  PR[GP1:91,1] = PR[GP1:90,1] + -54.611;
   1:  PR[GP1:91,2] = PR[GP1:90,2] + -30.612;
   1:L PR[91] 10mm/sec CNT100;
   1:  PR[GP1:91,1] = PR[GP1:90,1] + -47.452;
   1:  PR[GP1:91,2] = PR[GP1:90,2] + -32.843;
   1:L PR[91] 10mm/sec CNT100;
   1:  PR[GP1:91,1] = PR[GP1:90,1] + -42.540;
   1:  PR[GP1:91,2] = PR[GP1:90,2] + -34.146;
   1:L PR[91] 10mm/sec CNT100;
   1:  PR[GP1:91,1] = PR[GP1:90,1] + -32.956;
   1:  PR[GP1:91,2] = PR[GP1:90,2] + -33.612;
   1:L PR[91] 10mm/sec CNT100;
   1:  PR[GP1:91,1] = PR[GP1:90,1] + -30.132;
   1:  PR[GP1:91,2] = PR[GP1:90,2] + -33.296;
   1:L PR[91] 10mm/sec CNT100;
   1:  PR[GP1:91,1] = PR[GP1:90,1] + -19.213;
   1:  PR[GP1:91,2] = PR[GP1:90,2] + -28.502;
   1:L PR[91] 10mm/sec CNT100;
   1:  PR[GP1:91,1] = PR[GP1:90,1] + -18.911;
   1:  PR[GP1:91,2] = PR[GP1:90,2] + -28.344;
   1:L PR[91] 10mm/sec CNT100;
   1:  PR[GP1:91,1] = PR[GP1:90,1] + -17.107;
   1:  PR[GP1:91,2] = PR[GP1:90,2] + -26.580;
   1:L PR[91] 10mm/sec CNT100;
   1:  PR[GP1:91,1] = PR[GP1:90,1] + -10.026;
   1:  PR[GP1:91,2] = PR[GP1:90,2] + -19.923;
   1:L PR[91] 10mm/sec CNT100;
   1:  PR[GP1:91,1] = PR[GP1:90,1] + -9.145;
   1:  PR[GP1:91,2] = PR[GP1:90,2] + -18.468;
   1:L PR[91] 10mm/sec CNT100;
   1:  PR[GP1:91,1] = PR[GP1:90,1] + -4.436;
   1:  PR[GP1:91,2] = PR[GP1:90,2] + -8.658;
   1:L PR[91] 10mm/sec CNT100;
   1:  PR[GP1:91,1] = PR[GP1:90,1] + 3.921;
   1:L PR[91] 10mm/sec CNT100;
   1:  PR[GP1:91,1] = PR[GP1:90,1] + 8.001;
   1:  PR[GP1:91,2] = PR[GP1:90,2] + -17.702;
   1:  PR[GP1:91,3] = PR[GP1:90,3] + 24.705;
   1:L PR[91] 10mm/sec CNT100;
   1:  PR[GP1:91,1] = PR[GP1:90,1] + 9.477;
   1:  PR[GP1:91,2] = PR[GP1:90,2] + -20.138;
   1:L PR[91] 10mm/sec CNT100;
   1:  PR[GP1:91,1] = PR[GP1:90,1] + 17.926;
   1:  PR[GP1:91,2] = PR[GP1:90,2] + -28.101;
   1:L PR[91] 10mm/sec CNT100;
   1:  PR[GP1:91,1] = PR[GP1:90,1] + 18.361;
   1:  PR[GP1:91,2] = PR[GP1:90,2] + -28.449;
   1:L PR[91] 10mm/sec CNT100;
   1:  PR[GP1:91,1] = PR[GP1:90,1] + 20.903;
   1:  PR[GP1:91,2] = PR[GP1:90,2] + -29.509;
   1:L PR[91] 10mm/sec CNT100;
   1:  PR[GP1:91,1] = PR[GP1:90,1] + 29.656;
   1:  PR[GP1:91,2] = PR[GP1:90,2] + -33.352;
   1:L PR[91] 10mm/sec CNT100;
   1:  PR[GP1:91,1] = PR[GP1:90,1] + 31.498;
   1:  PR[GP1:91,2] = PR[GP1:90,2] + -33.559;
   1:L PR[91] 10mm/sec CNT100;
   1:  PR[GP1:91,1] = PR[GP1:90,1] + 42.040;
   1:  PR[GP1:91,2] = PR[GP1:90,2] + -34.151;
   1:L PR[91] 10mm/sec CNT100;
   1:  PR[GP1:91,1] = PR[GP1:90,1] + 46.087;
   1:  PR[GP1:91,2] = PR[GP1:90,2] + -33.078;
   1:L PR[91] 10mm/sec CNT100;
   1:  PR[GP1:91,1] = PR[GP1:90,1] + 54.078;
   1:  PR[GP1:91,2] = PR[GP1:90,2] + -30.589;
   1:L PR[91] 10mm/sec CNT100;
   1:  PR[GP1:91,1] = PR[GP1:90,1] + 58.899;
   1:  PR[GP1:91,2] = PR[GP1:90,2] + -27.066;
   1:L PR[91] 10mm/sec CNT100;
   1:  PR[GP1:91,1] = PR[GP1:90,1] + 64.165;
   1:  PR[GP1:91,2] = PR[GP1:90,2] + -22.969;
   1:L PR[91] 10mm/sec CNT100;
   1:  PR[GP1:91,1] = PR[GP1:90,1] + 67.981;
   1:  PR[GP1:91,2] = PR[GP1:90,2] + -16.951;
   1:L PR[91] 10mm/sec CNT100;
   1:  PR[GP1:91,1] = PR[GP1:90,1] + 70.875;
   1:  PR[GP1:91,2] = PR[GP1:90,2] + -12.198;
   1:L PR[91] 10mm/sec CNT100;
   1:  PR[GP1:91,1] = PR[GP1:90,1] + 72.360;
   1:  PR[GP1:91,2] = PR[GP1:90,2] + -4.452;
   1:L PR[91] 10mm/sec CNT100;
   1:  PR[GP1:91,1] = PR[GP1:90,1] + 73.233;
   1:  PR[GP1:91,2] = PR[GP1:90,2] + 0.277;
   1:L PR[91] 10mm/sec CNT100;
   1:  PR[GP1:91,1] = PR[GP1:90,1] + 71.774;
   1:  PR[GP1:91,2] = PR[GP1:90,2] + 7.873;
   1:L PR[91] 10mm/sec CNT100;
   1:  PR[GP1:91,1] = PR[GP1:90,1] + 70.873;
   1:  PR[GP1:91,2] = PR[GP1:90,2] + 12.758;
   1:L PR[91] 10mm/sec CNT100;
   1:  PR[GP1:91,1] = PR[GP1:90,1] + 67.981;
   1:  PR[GP1:91,2] = PR[GP1:90,2] + 17.510;
   1:L PR[91] 10mm/sec CNT100;
   1:  PR[GP1:91,1] = PR[GP1:90,1] + 64.165;
   1:  PR[GP1:91,2] = PR[GP1:90,2] + 23.527;
   1:L PR[91] 10mm/sec CNT100;
   1:  PR[GP1:91,1] = PR[GP1:90,1] + 58.899;
   1:  PR[GP1:91,2] = PR[GP1:90,2] + 27.624;
   1:L PR[91] 10mm/sec CNT100;
   1:  PR[GP1:91,1] = PR[GP1:90,1] + 54.078;
   1:  PR[GP1:91,2] = PR[GP1:90,2] + 31.147;
   1:L PR[91] 10mm/sec CNT100;
   1:  PR[GP1:91,1] = PR[GP1:90,1] + 46.087;
   1:  PR[GP1:91,2] = PR[GP1:90,2] + 33.636;
   1:L PR[91] 10mm/sec CNT100;
   1:  PR[GP1:91,1] = PR[GP1:90,1] + 42.039;
   1:  PR[GP1:91,2] = PR[GP1:90,2] + 34.709;
   1:L PR[91] 10mm/sec CNT100;
   1:  PR[GP1:91,1] = PR[GP1:90,1] + 31.498;
   1:  PR[GP1:91,2] = PR[GP1:90,2] + 34.117;
   1:L PR[91] 10mm/sec CNT100;
   1:  PR[GP1:91,1] = PR[GP1:90,1] + 29.656;
   1:  PR[GP1:91,2] = PR[GP1:90,2] + 33.910;
   1:L PR[91] 10mm/sec CNT100;
   1:  PR[GP1:91,1] = PR[GP1:90,1] + 20.903;
   1:  PR[GP1:91,2] = PR[GP1:90,2] + 30.067;
   1:L PR[91] 10mm/sec CNT100;
   1:  PR[GP1:91,1] = PR[GP1:90,1] + 18.361;
   1:  PR[GP1:91,2] = PR[GP1:90,2] + 29.007;
   1:L PR[91] 10mm/sec CNT100;
   1:  PR[GP1:91,1] = PR[GP1:90,1] + 17.926;
   1:  PR[GP1:91,2] = PR[GP1:90,2] + 28.659;
   1:L PR[91] 10mm/sec CNT100;
   1:  PR[GP1:91,1] = PR[GP1:90,1] + 9.477;
   1:  PR[GP1:91,2] = PR[GP1:90,2] + 20.696;
   1:L PR[91] 10mm/sec CNT100;
   1:  PR[GP1:91,1] = PR[GP1:90,1] + 8.001;
   1:  PR[GP1:91,2] = PR[GP1:90,2] + 18.260;
   1:L PR[91] 10mm/sec CNT100;
   1:  PR[GP1:91,1] = PR[GP1:90,1] + 3.811;
   1:  PR[GP1:91,2] = PR[GP1:90,2] + 9.541;
   1:L PR[91] 10mm/sec CNT100;
   1:  PR[GP1:91,1] = PR[GP1:90,1] + -4.358;
   1:L PR[91] 10mm/sec CNT100;
   1:  PR[GP1:91,1] = PR[GP1:90,1] + -8.538;
   1:  PR[GP1:91,2] = PR[GP1:90,2] + 18.281;
   1:L PR[91] 10mm/sec CNT100;
   1:  PR[GP1:91,1] = PR[GP1:90,1] + -10.013;
   1:  PR[GP1:91,2] = PR[GP1:90,2] + 20.718;
   1:L PR[91] 10mm/sec CNT100;
   1:  PR[GP1:91,1] = PR[GP1:90,1] + -18.467;
   1:  PR[GP1:91,2] = PR[GP1:90,2] + 28.666;
   1:L PR[91] 10mm/sec CNT100;
   1:  PR[GP1:91,1] = PR[GP1:90,1] + -18.900;
   1:  PR[GP1:91,2] = PR[GP1:90,2] + 29.011;
   1:L PR[91] 10mm/sec CNT100;
   1:  PR[GP1:91,1] = PR[GP1:90,1] + -21.430;
   1:  PR[GP1:91,2] = PR[GP1:90,2] + 30.067;
   1:L PR[91] 10mm/sec CNT100;
   1:  PR[GP1:91,1] = PR[GP1:90,1] + -30.193;
   1:  PR[GP1:91,2] = PR[GP1:90,2] + 33.914;
   1:L PR[91] 10mm/sec CNT100;
   1:  PR[GP1:91,1] = PR[GP1:90,1] + -32.038;
   1:  PR[GP1:91,2] = PR[GP1:90,2] + 34.120;
   1:L PR[91] 10mm/sec CNT100;
   1:  PR[GP1:91,1] = PR[GP1:90,1] + -42.574;
   1:  PR[GP1:91,2] = PR[GP1:90,2] + 34.708;
   1:L PR[91] 10mm/sec CNT100;
   1:  PR[GP1:91,1] = PR[GP1:90,1] + -46.622;
   1:  PR[GP1:91,2] = PR[GP1:90,2] + 33.634;
   1:L PR[91] 10mm/sec CNT100;
   1:  PR[GP1:91,1] = PR[GP1:90,1] + -54.610;
   1:  PR[GP1:91,2] = PR[GP1:90,2] + 31.144;
   1:L PR[91] 10mm/sec CNT100;
   1:  PR[GP1:91,1] = PR[GP1:90,1] + -59.430;
   1:  PR[GP1:91,2] = PR[GP1:90,2] + 27.621;
   1:L PR[91] 10mm/sec CNT100;
   1:  PR[GP1:91,1] = PR[GP1:90,1] + -64.694;
   1:  PR[GP1:91,2] = PR[GP1:90,2] + 23.526;
   1:L PR[91] 10mm/sec CNT100;
   1:  PR[GP1:91,1] = PR[GP1:90,1] + -68.509;
   1:  PR[GP1:91,2] = PR[GP1:90,2] + 17.507;
   1:L PR[91] 10mm/sec CNT100;
   1:  PR[GP1:91,1] = PR[GP1:90,1] + -71.402;
   1:  PR[GP1:91,2] = PR[GP1:90,2] + 12.749;
   1:L PR[91] 10mm/sec CNT100;
   1:  PR[GP1:91,1] = PR[GP1:90,1] + -72.887;
   1:  PR[GP1:91,2] = PR[GP1:90,2] + 5.005;
   1:L PR[91] 10mm/sec CNT100;
   1:  PR[GP1:91,1] = PR[GP1:90,1] + -73.760;
   1:  PR[GP1:91,2] = PR[GP1:90,2] + 0.281;
   1:L PR[91] 10mm/sec CNT100;
   1:  PR[GP1:91,1] = PR[GP1:90,1] + -72.301;
   1:  PR[GP1:91,2] = PR[GP1:90,2] + -7.313;
   1:L PR[91] 10mm/sec CNT100;
   1:  PR[GP1:91,1] = PR[GP1:90,1] + -71.400;
   1:  PR[GP1:91,2] = PR[GP1:90,2] + -12.193;
   1:L PR[91] 10mm/sec CNT100;
   1:  PR[GP1:91,1] = PR[GP1:90,1] + -68.509;
   1:  PR[GP1:91,2] = PR[GP1:90,2] + -16.949;
   1:L PR[91] 10mm/sec CNT100;
   1:  PR[GP1:91,1] = PR[GP1:90,1] + -64.694;
   1:  PR[GP1:91,2] = PR[GP1:90,2] + -22.968;
   1:L PR[91] 10mm/sec CNT100;
   1:  PR[GP1:91,1] = PR[GP1:90,1] + -59.430;
   1:  PR[GP1:91,2] = PR[GP1:90,2] + -27.063;
   1:L PR[91] 10mm/sec CNT100;
   1:  PR[GP1:91,1] = PR[GP1:90,1] + -54.609;
   1:  PR[GP1:91,2] = PR[GP1:90,2] + -30.586;
   1:L PR[91] 10mm/sec CNT100;
   1:  PR[GP1:91,1] = PR[GP1:90,1] + -46.622;
   1:  PR[GP1:91,2] = PR[GP1:90,2] + -33.076;
   1:L PR[91] 10mm/sec CNT100;
   1:  PR[GP1:91,1] = PR[GP1:90,1] + -42.574;
   1:  PR[GP1:91,2] = PR[GP1:90,2] + -34.150;
   1:L PR[91] 10mm/sec CNT100;
   1:  PR[GP1:91,1] = PR[GP1:90,1] + -32.038;
   1:  PR[GP1:91,2] = PR[GP1:90,2] + -33.562;
   1:L PR[91] 10mm/sec CNT100;
   1:  PR[GP1:91,1] = PR[GP1:90,1] + -30.193;
   1:  PR[GP1:91,2] = PR[GP1:90,2] + -33.356;
   1:L PR[91] 10mm/sec CNT100;
   1:  PR[GP1:91,1] = PR[GP1:90,1] + -21.430;
   1:  PR[GP1:91,2] = PR[GP1:90,2] + -29.509;
   1:L PR[91] 10mm/sec CNT100;
   1:  PR[GP1:91,1] = PR[GP1:90,1] + -18.900;
   1:  PR[GP1:91,2] = PR[GP1:90,2] + -28.453;
   1:L PR[91] 10mm/sec CNT100;
   1:  PR[GP1:91,1] = PR[GP1:90,1] + -18.467;
   1:  PR[GP1:91,2] = PR[GP1:90,2] + -28.108;
   1:L PR[91] 10mm/sec CNT100;
   1:  PR[GP1:91,1] = PR[GP1:90,1] + -10.013;
   1:  PR[GP1:91,2] = PR[GP1:90,2] + -20.160;
   1:L PR[91] 10mm/sec CNT100;
   1:  PR[GP1:91,1] = PR[GP1:90,1] + -8.538;
   1:  PR[GP1:91,2] = PR[GP1:90,2] + -17.723;
   1:L PR[91] 10mm/sec CNT100;
   1:  PR[GP1:91,1] = PR[GP1:90,1] + -4.343;
   1:  PR[GP1:91,2] = PR[GP1:90,2] + -8.983;
   1:L PR[91] 10mm/sec CNT100;
   1:  PR[GP1:91,1] = PR[GP1:90,1] + 3.825;
   1:L PR[91] 10mm/sec CNT100;
   1:  PR[GP1:91,1] = PR[GP1:90,1] + 7.394;
   1:  PR[GP1:91,2] = PR[GP1:90,2] + -16.960;
   1:  PR[GP1:91,3] = PR[GP1:90,3] + 25.315;
   1:L PR[91] 10mm/sec CNT100;
   1:  PR[GP1:91,1] = PR[GP1:90,1] + 9.465;
   1:  PR[GP1:91,2] = PR[GP1:90,2] + -20.375;
   1:L PR[91] 10mm/sec CNT100;
   1:  PR[GP1:91,1] = PR[GP1:90,1] + 17.053;
   1:  PR[GP1:91,2] = PR[GP1:90,2] + -27.527;
   1:L PR[91] 10mm/sec CNT100;
   1:  PR[GP1:91,1] = PR[GP1:90,1] + 18.379;
   1:  PR[GP1:91,2] = PR[GP1:90,2] + -28.588;
   1:L PR[91] 10mm/sec CNT100;
   1:  PR[GP1:91,1] = PR[GP1:90,1] + 25.402;
   1:  PR[GP1:91,2] = PR[GP1:90,2] + -31.518;
   1:L PR[91] 10mm/sec CNT100;
   1:  PR[GP1:91,1] = PR[GP1:90,1] + 29.717;
   1:  PR[GP1:91,2] = PR[GP1:90,2] + -33.412;
   1:L PR[91] 10mm/sec CNT100;
   1:  PR[GP1:91,1] = PR[GP1:90,1] + 30.579;
   1:  PR[GP1:91,2] = PR[GP1:90,2] + -33.509;
   1:L PR[91] 10mm/sec CNT100;
   1:  PR[GP1:91,1] = PR[GP1:90,1] + 42.073;
   1:  PR[GP1:91,2] = PR[GP1:90,2] + -34.155;
   1:L PR[91] 10mm/sec CNT100;
   1:  PR[GP1:91,1] = PR[GP1:90,1] + 45.256;
   1:  PR[GP1:91,2] = PR[GP1:90,2] + -33.310;
   1:L PR[91] 10mm/sec CNT100;
   1:  PR[GP1:91,1] = PR[GP1:90,1] + 54.076;
   1:  PR[GP1:91,2] = PR[GP1:90,2] + -30.564;
   1:L PR[91] 10mm/sec CNT100;
   1:  PR[GP1:91,1] = PR[GP1:90,1] + 58.242;
   1:  PR[GP1:91,2] = PR[GP1:90,2] + -27.520;
   1:L PR[91] 10mm/sec CNT100;
   1:  PR[GP1:91,1] = PR[GP1:90,1] + 64.130;
   1:  PR[GP1:91,2] = PR[GP1:90,2] + -22.939;
   1:L PR[91] 10mm/sec CNT100;
   1:  PR[GP1:91,1] = PR[GP1:90,1] + 67.546;
   1:  PR[GP1:91,2] = PR[GP1:90,2] + -17.551;
   1:L PR[91] 10mm/sec CNT100;
   1:  PR[GP1:91,1] = PR[GP1:90,1] + 70.817;
   1:  PR[GP1:91,2] = PR[GP1:90,2] + -12.179;
   1:L PR[91] 10mm/sec CNT100;
   1:  PR[GP1:91,1] = PR[GP1:90,1] + 72.167;
   1:  PR[GP1:91,2] = PR[GP1:90,2] + -5.137;
   1:L PR[91] 10mm/sec CNT100;
   1:  PR[GP1:91,1] = PR[GP1:90,1] + 73.167;
   1:  PR[GP1:91,2] = PR[GP1:90,2] + 0.277;
   1:L PR[91] 10mm/sec CNT100;
   1:  PR[GP1:91,1] = PR[GP1:90,1] + 71.834;
   1:  PR[GP1:91,2] = PR[GP1:90,2] + 7.217;
   1:L PR[91] 10mm/sec CNT100;
   1:  PR[GP1:91,1] = PR[GP1:90,1] + 70.816;
   1:  PR[GP1:91,2] = PR[GP1:90,2] + 12.739;
   1:L PR[91] 10mm/sec CNT100;
   1:  PR[GP1:91,1] = PR[GP1:90,1] + 67.546;
   1:  PR[GP1:91,2] = PR[GP1:90,2] + 18.109;
   1:L PR[91] 10mm/sec CNT100;
   1:  PR[GP1:91,1] = PR[GP1:90,1] + 64.130;
   1:  PR[GP1:91,2] = PR[GP1:90,2] + 23.497;
   1:L PR[91] 10mm/sec CNT100;
   1:  PR[GP1:91,1] = PR[GP1:90,1] + 58.242;
   1:  PR[GP1:91,2] = PR[GP1:90,2] + 28.078;
   1:L PR[91] 10mm/sec CNT100;
   1:  PR[GP1:91,1] = PR[GP1:90,1] + 54.076;
   1:  PR[GP1:91,2] = PR[GP1:90,2] + 31.122;
   1:L PR[91] 10mm/sec CNT100;
